(* Read only; Axis ID of the linked NC Axis *)
PROPERTY NcAxisId : UDINT
GET
NcAxisId := _AxisRef.NcToPlc.AxisId;
END_GET
END_PROPERTY

(* Read only; Axis ID of the linked NC Axis *)
PROPERTY NcAxisName : String(31)
GET
 NcAxisName := stAxisName;
END_GET
END_PROPERTY

METHOD ParamCheck : BOOL;
VAR_INST
  bTmp      : Bool;
  res       : Tc2_MC2.ST_McOutputs;
  nState    : DINT;
  stParaNr  : Tc2_MC2.MC_AxisParameter;
END_VAR

CASE nState 
OF
  0:
    ReadParameter(FALSE, stParaNr);
    bTmp              := FALSE;
    nState            := 1;
END_CASE
CASE nState 
OF
  1:
    IF NOT stDefaultAcceleration.bValid 
    THEN
      stParaNr        := AxisAcc;
      nState          := 10;

    ELSIF NOT stDefaultDeceleration.bValid 
    THEN
      stParaNr        := AxisDec;
      nState          := 10;

    ELSIF NOT stDefaultJerk.bValid 
    THEN
      stParaNr        := AxisJerk;
      nState          := 10;

    ELSIF NOT stHomingSearchVelo.bValid 
    THEN
      stParaNr        := AxisCalibrationVelocityForward;
      nState          := 10;

    ELSIF NOT stHomingVelo.bValid 
    THEN
      stParaNr        := AxisCalibrationVelocityBackward;
      nState          := 10;

    ELSIF NOT stMaxAcceleration.bValid 
    THEN
      stParaNr        := AxisMaximumAcceleration;
      nState          := 10;

    ELSIF NOT stMaxDeceleration.bValid 
    THEN
      stParaNr        := AxisMaximumDeceleration;
      nState          := 10;

    ELSIF NOT stMaxVelocity.bValid 
    THEN
      stParaNr        := AxisVeloMax;
      nState          := 10;

    ELSIF NOT stSwPosLimitNegative.bValid 
    THEN
      stParaNr        := AxisMinSoftPosLimit;
      nState          := 10;

    ELSIF NOT stSwPosLimitNegativeActive.bValid 
    THEN
      stParaNr        := AxisEnMinSoftPosLimit;
      nState          := 10;

    ELSIF NOT stSwPosLimitPositive.bValid 
    THEN
      stParaNr        := AxisMaxSoftPosLimit;
      nState          := 10;

    ELSIF NOT stSwPosLimitPositiveActive.bValid 
    THEN
      stParaNr        := AxisEnMaxSoftPosLimit;
      nState          := 10;

    ELSIF NOT stTargetPositionWindow.bValid 
    THEN
      stParaNr        := AxisTargetPositionWindow;
      nState          := 10;

    ELSE
      fbGetCurTaskIndex();
      _rCycleTime     := UDINT_TO_LREAL(_TaskInfo[fbGetCurTaskIndex.index].CycleTime)/10000.0;

      bTmp            := TRUE; // done
    END_IF
END_CASE
CASE nState 
OF
  10:
    bTmp              := FALSE;
    res               := ReadParameter(FALSE, stParaNr);
    nState            := 20;
END_CASE
CASE nState 
OF
  20:
    res               := ReadParameter(TRUE, stParaNr);
    IF res.Done
    THEN
      nState          := 30;
    END_IF

END_CASE
CASE nState 
OF
  30:
    nState                                := 0;
    CASE stParaNr 
    OF
      AxisEnMinSoftPosLimit: 
        stSwPosLimitNegativeActive.bValue := LREAL_TO_BOOL(fbReadParameter.Value);
        stSwPosLimitNegativeActive.bValid := TRUE;
    
      AxisEnMaxSoftPosLimit: 
        stSwPosLimitPositiveActive.bValue := LREAL_TO_BOOL(fbReadParameter.Value);
        stSwPosLimitPositiveActive.bValid := TRUE;
    
      AxisAcc: 
        stDefaultAcceleration.fValue      := fReadParamValue;
        stDefaultAcceleration.bValid      := TRUE;

      AxisDec: 
        stDefaultDeceleration.fValue      := fReadParamValue;
        stDefaultDeceleration.bValid      := TRUE;

      AxisJerk: 
        stDefaultJerk.fValue              := fReadParamValue;
        stDefaultJerk.bValid              := TRUE;

      AxisMaximumAcceleration : 
        stMaxAcceleration.fValue          := fReadParamValue;
        stMaxAcceleration.bValid          := TRUE;

      AxisMaximumDeceleration: 
        stMaxDeceleration.fValue          := fReadParamValue;
        stMaxDeceleration.bValid          := TRUE;

      AxisVeloMax: 
        stMaxVelocity.fValue              := fReadParamValue;
        fDefaultVelocity                  := stMaxVelocity.fValue * 0.1;
        stMaxVelocity.bValid              := TRUE;

      AxisMinSoftPosLimit: 
        stSwPosLimitNegative.fValue       := fReadParamValue;
        stSwPosLimitNegative.bValid       := TRUE;

      AxisMaxSoftPosLimit: 
        stSwPosLimitPositive.fValue       := fReadParamValue;
        stSwPosLimitPositive.bValid       := TRUE;

      AxisCalibrationVelocityForward: 
        stHomingSearchVelo.fValue         := fReadParamValue;
        stHomingSearchVelo.bValid         := TRUE;

      AxisCalibrationVelocityBackward: 
        stHomingVelo.fValue               := fReadParamValue;
        stHomingVelo.bValid               := TRUE;

      AxisTargetPositionWindow:
        stTargetPositionWindow.fValue     := fReadParamValue;
        stTargetPositionWindow.bValid     := TRUE;

    END_CASE

END_CASE

ParamCheck := bTmp;
END_METHOD

PROPERTY pAxisRef : POINTER TO AXIS_REF
GET
pAxisRef := ADR(_AxisRef);
END_GET
END_PROPERTY

PROPERTY Position : LREAL
GET
Position := _AxisRef.NcToPlc.ActPos;
END_GET
END_PROPERTY

{attribute '''NORMAL__COMMENT' := ' Will try to read a parameter from the NC axis; If the value is read, the Value is available at the ReadParamValue property.
  Refer to MC_ReadParameter Function Block in the Tc2_MC2 library; READMODE_ONCE is used as ReadMode '}
(* Will try to read a parameter from the NC axis; If the value is read, the Value is available at the ReadParamValue property.
  Refer to MC_ReadParameter Function Block in the Tc2_MC2 library; READMODE_ONCE is used as ReadMode *)
METHOD ReadParameter : Tc2_MC2.ST_McOutputs
VAR_INPUT
  Execute           : BOOL;
  (* Number of the parameter to be read. Refer to the MC_AxisParameter type defined at Tc2_MC2 library *)
  {attribute '''NORMAL__COMMENT' := ' Number of the parameter to be read. Refer to the MC_AxisParameter type defined at Tc2_MC2 library '}
  ParameterNumber   : Tc2_MC2.MC_AxisParameter;
END_VAR
VAR_INST
  res               : Tc2_MC2.ST_McOutputs;
  nState            : DINT;
END_VAR

CASE nState OF
  0:
    IF Execute
    THEN
      memset(ADR(res),0,SIZEOF(res));
      res.Busy                          := TRUE;

      fbReadParameter.ParameterNumber   := ParameterNumber;
      fbReadParameter.Enable            := FALSE;

      nState                            := 10;
    END_IF
END_CASE
CASE nState OF
  10:
    fbReadParameter.Enable              := TRUE;

    IF fbReadParameter.Valid
    THEN
      fbReadParameter.Enable            := FALSE;
      nState                            := 20;
    ELSE
      IF fbReadParameter.Error
      THEN
        res.ErrorID                     := fbWriteParameter.ErrorID;

        stMsg.eType                     := E_MessageType.eMessageError;
        stMsg.eDevice                   := e_Device.Axis + TO_DINT(_AxisRef.NcToPlc.AxisId);
        stMsg.eSubdevice                := e_SubDevice.fbReadParameter;
        stMsg.iErrorNumber              := fbReadParameter.ErrorID;

        f_MessageSet(stMsg);
        MsgAdd(stMsg);

        fbReadParameter.Enable          := FALSE;
        nState                          := 99;
      END_IF
    END_IF
END_CASE
CASE nState OF
  20:
    res.Busy                            := FALSE;
    res.Done                            := TRUE;

  99:
    res.Busy                            := FALSE;
    res.Error                           := TRUE;
END_CASE

fbReadParameter(Axis                    := _AxisRef, 
                ParameterNumber         := ParameterNumber, 
                ReadMode                := Tc2_MC2.READMODE_ONCE, 
                Value                   => fReadParamValue);

IF NOT Execute
THEN
  memset(ADR(res),0,SIZEOF(res));
  nState                                := 0;
END_IF

ReadParameter := res;
END_METHOD

(* Read only; Returns the value from the last successful read by ReadParameter methode *)
PROPERTY ReadParamValue : LREAL
GET
ReadParamValue := fReadParamValue;
END_GET
END_PROPERTY

(* Speed override factor in percent [%] to all movements. Refer to MC_Power Function Block in the Tc2_MC2 library *)
PROPERTY SpeedOverride : LREAL
GET
SpeedOverride := fbPower.Override;
END_GET
SET
fbPower.Override := SpeedOverride;
END_SET
END_PROPERTY

PROPERTY StartUpDone : BOOL
GET
StartUpDone := _bStartUp;
END_GET
END_PROPERTY

PROPERTY StartUpError : Bool
GET
StartUpError := _bStartUpError;
END_GET
END_PROPERTY

(* Read only; Initiates read the actual Axis status; returns the Status of the last performed read *) 
PROPERTY Status : Tc2_MC2.ST_AxisStatus
GET
Status := _AxisRef.Status;
END_GET
END_PROPERTY

METHOD Stop : Tc2_MC2.ST_McOutputs
VAR_INPUT
  Execute   : BOOL;
END_VAR
VAR_INST
  res       : Tc2_MC2.ST_McOutputs;
  nState    : DINT;
  fUsedDec,
  fUsedJerk : LREAL;
  itmp      : DINT;
END_VAR
CASE nState OF
  0:
    IF Execute
    THEN
      memset(ADR(res),0,SIZEOF(res));
      memset(ADR(itmp),0,SIZEOF(itmp));
      res.Busy                := TRUE;

      fUsedDec                := stDefaultDeceleration.fValue;
      fUsedJerk               := stDefaultJerk.fValue;

      fbStop(Axis             := _AxisRef,  
             Execute          := FALSE, 
             Deceleration     := fUsedDec, 
             Jerk             := fUsedJerk);

      fbReset(Axis            := _AxisRef, 
              Execute         := FALSE);

      nState := 10;
    END_IF
END_CASE
CASE nState OF
  10:
    fbStop(Axis               := _AxisRef, 
           Execute            := TRUE);

    IF fbStop.Done
    THEN
      fbStop(Axis             := _AxisRef, 
             Execute          := FALSE);

      nState := 20;

    ELSE
      IF fbStop.Error
      THEN
        res.ErrorID           := fbStop.ErrorID;

        stMsg.eType           := E_MessageType.eMessageError;
        stMsg.eDevice         := e_Device.Axis + UDINT_TO_DINT(_AxisRef.NcToPlc.AxisId);
        stMsg.eSubdevice      := e_SubDevice.fbStop;
        stMsg.iErrorNumber    := fbStop.ErrorID;
        f_MessageSet(stMsg);
        MsgAdd(stMsg);

        fbReset(Axis          := _AxisRef, 
                Execute       := TRUE);

        nState := 98;

      ELSIF NOT _AxisRef.Status.Stopping
      THEN
        itmp := itmp +1;
        // todo: faststop?
      END_IF
    END_IF
END_CASE
CASE nState OF
  20:
    res.Busy := FALSE;
    res.Done := TRUE;

  98:
    fbStop(Axis               := _AxisRef, 
           Execute            := FALSE);

    fbReset(Axis              := _AxisRef, 
            Execute           := FALSE);
    nState := 99;

END_CASE
CASE nState OF
  99:
    res.Busy                  := FALSE;
    res.Error                 := TRUE;
END_CASE

IF NOT Execute
THEN
  memset(ADR(res),0,SIZEOF(res));
  nState                      := 0;
END_IF

Stop := res;
END_METHOD

PROPERTY Version : STRING
(* ToDo:
- Testen
*)
GET
Version := '1.0';
(*
  0.1   09.2016 MR  Erste Version des Achsbausteins als OOP Wrapper der MC Bausteine; Die Funktionen können meißt (Außnahme: Jog) durch einen einmaliger Methodenaufruf angestossen werden;
            der weitere Aufruf erfolgt dann automatisch über den zyklischen Aufruf der FB Instanz und die interne Methode CyclicCallOnBusy. Die FB Instanz muss immer zyklisch 
            aufgerufen werden.
            
  1.0
  2022 06 30
  HAUD
  - 
  - cyclic method calls required
  - motion methods contain VAR_INST (fixed procedure, no race conditions)
  - Motion Parameter as properties (input from stCtrl by AxisController)
  - cyclic ca

*)
END_GET
END_PROPERTY

{attribute '''NORMAL__COMMENT' := ' Will try to write a parameter from the NC axis; Refer to MC_WriteParameter Function Block in the Tc2_MC2 library '}
(* Will try to write a parameter from the NC axis; Refer to MC_WriteParameter Function Block in the Tc2_MC2 library *)
METHOD WriteParameter : Tc2_MC2.ST_McOutputs
VAR_INPUT
  Execute   : BOOL;
  (* Number of the parameter to be written. Refer to the MC_AxisParameter type defined at Tc2_MC2 library *)
  {attribute '''NORMAL__COMMENT' := ' Number of the parameter to be written. Refer to the MC_AxisParameter type defined at Tc2_MC2 library '}
  ParameterNumber : Tc2_MC2.MC_AxisParameter;
  (* defines the value to be written to the parameter *)
  {attribute '''NORMAL__COMMENT' := ' defines the value to be written to the parameter '}
  Value : LREAL;
END_VAR
VAR_INST
  res       : Tc2_MC2.ST_McOutputs;
  nState    : DINT;
END_VAR

CASE nState OF
  0:
    IF Execute
    THEN
      memset(ADR(res),0,SIZEOF(res));

      res.Busy                                := TRUE;

      fbWriteParameter.ParameterNumber        := ParameterNumber;

      fbWriteParameter(Axis                   := _AxisRef, 
                       Execute                := FALSE);
 
      nState                                  := 10;
    END_IF
END_CASE
CASE nState OF
  10:
    fbWriteParameter.Execute                  := TRUE;

    IF fbWriteParameter.Done
    THEN
      nState                                  := 20;

      CASE fbWriteParameter.ParameterNumber 
      OF
        AxisEnMinSoftPosLimit: 
          stSwPosLimitNegativeActive.bValue   := TO_BOOL(Value);

        AxisEnMaxSoftPosLimit: 
          stSwPosLimitPositiveActive.bValue   := TO_BOOL(Value);

        AxisAcc: 
          stDefaultAcceleration.fValue        := Value;

        AxisDec: 
          stDefaultDeceleration.fValue        := Value;

        AxisJerk: 
          stDefaultJerk.fValue                := Value;

        AxisMaximumAcceleration : 
          stMaxAcceleration.fValue            := Value;

        AxisMaximumDeceleration: 
          stMaxDeceleration.fValue            := Value;

        AxisVeloMax: 
          stMaxVelocity.fValue                := Value;

        AxisMinSoftPosLimit: 
          stSwPosLimitNegative.fValue         := Value;

        AxisMaxSoftPosLimit: 
          stSwPosLimitPositive.fValue         := Value;

        AxisCalibrationVelocityForward: 
          stHomingSearchVelo.fValue           := Value;

        AxisCalibrationVelocityBackward: 
          stHomingVelo.fValue                 := Value;

        AxisTargetPositionWindow:
          stTargetPositionWindow.fValue       := Value;
      END_CASE
    ELSE
      IF fbWriteParameter.Error
      THEN
        res.Busy                              := FALSE;
        res.Error                             := TRUE;
        res.ErrorID                           := fbWriteParameter.ErrorID;

        stMsg.eType                           := E_MessageType.eMessageError;
        stMsg.eDevice                         := e_Device.Axis + TO_DINT(_AxisRef.NcToPlc.AxisId);
        stMsg.eSubdevice                      := e_SubDevice.fbWriteParameter;
        stMsg.iErrorNumber                    := fbWriteParameter.ErrorID;

        fbWriteParameter.Execute              := FALSE;

        f_MessageSet(stMsg);
        MsgAdd(stMsg);

        nState                                := 99;
      END_IF
    END_IF
END_CASE
CASE nState OF
  20:
    res.Busy                                  := FALSE;
    res.Done                                  := TRUE;

  99:
    res.Busy                                  := FALSE;
    res.Error                                 := TRUE;

END_CASE


IF NOT Execute
THEN
  memset(ADR(res),0,SIZEOF(res));

  fbWriteParameter.Execute                    := FALSE;
  nState                                      := 0;
END_IF


fbWriteParameter(Axis                         := _AxisRef, 
                 ParameterNumber              := ParameterNumber, 
                 Value                        := Value, 
                 Done                         => WriteParameter.Done, 
                 Busy                         => WriteParameter.Busy, 
                 Error                        => WriteParameter.Error, 
                 ErrorID                      => WriteParameter.ErrorID);


WriteParameter := res;
END_METHOD

END_FUNCTION_BLOCK

// ---- POUs/MSG/f_MessageSet.TcPOU
FUNCTION f_MessageSet : BOOL
VAR_INPUT
  stMessage   : ST_Message;
END_VAR
VAR
  uiIndex   : INT;
  uiFound   : INT;
END_VAR

stMessage.tTime := GVL_AXIS_CTRL.gsLocalTime;

FOR uiIndex := 1 TO GVL_AXIS_CTRL.gciMaxMessage
DO
  IF (GVL_AXIS_CTRL.gatMessages[uiIndex].eType = e_MessageType.eMessageEmpty)
  THEN
    GVL_AXIS_CTRL.gatMessages[uiIndex] := stMessage;
    GVL_AXIS_CTRL.giMsgIndex := uiIndex;
    EXIT;
  END_IF
END_FOR

IF (stMessage.eType = E_MessageType.eMessageError)
THEN
  GVL_AXIS_CTRL.giErrorIndex := GVL_AXIS_CTRL.giErrorIndex + 1;
END_IF

END_FUNCTION

// ---- POUs/_FunctionBlocks/fb_ResetSercos.TcPOU
FUNCTION_BLOCK fb_ResetSercos
VAR_INPUT
	bExecute  : BOOL;
	eDevice		: e_Device;
	p_AxisRef	: POINTER TO Tc2_MC2.AXIS_REF;
END_VAR
VAR_OUTPUT
	stMcOutput : ST_McOutputs;
END_VAR
VAR
	diStep			: DINT;
	tonDelay		: ton;
	_stMessage	: ST_Message;
	fbResetSercos		: FB_SoEReset;
	iRepeat			: INT;
END_VAR

IF NOT bExecute
THEN
	stMcOutput.Active := FALSE;
	stMcOutput.Done := FALSE;
	diStep := 0;
END_IF

IF bExecute AND diStep = 0
THEN
	diStep := 10;
END_IF

IF p_AxisRef = 0
THEN
	RETURN;
END_IF

CASE diStep OF

	0:
		iRepeat := 0;
		tonDelay(IN:= FALSE);
		fbResetSercos(
			NetId:= , 
			Execute:= FALSE, 
			Timeout:= , 
			Axis:= p_AxisRef^, 
			Busy=> , 
			Error=> , 
			AdsErrId=> , 
			SercosErrId=> );

	10:
		stMcOutput.Active := TRUE;
		tonDelay(PT:= T#1500MS, IN:= TRUE);
		fbResetSercos(
			NetId:= , 
			Execute:= TRUE, 
			Timeout:= , 
			Axis:= p_AxisRef^, 
			Busy=> , 
			Error=> , 
			AdsErrId=> , 
			SercosErrId=> );

		IF NOT fbResetSercos.Busy
		THEN
			diStep := 20;
		END_IF

		IF tonDelay.Q AND p_AxisRef^.NcToPlc.StateDWord.28
		THEN
			iRepeat := iRepeat + 1;
			tonDelay(IN:= FALSE);
			fbResetSercos(
				NetId:= , 
				Execute:= FALSE, 
				Timeout:= , 
				Axis:= p_AxisRef^, 
				Busy=> , 
				Error=> , 
				AdsErrId=> , 
				SercosErrId=> );
		END_IF
 

	20:
		stMcOutput.Done := TRUE;

		IF NOT bExecute
		THEN
			fbResetSercos(Execute:= FALSE, Axis:= p_AxisRef^);
			memset(ADR(stMcOutput), 0, SIZEOF(stMcOutput));
			diStep :=0;
		END_IF
END_CASE

stMcOutput.Busy 		:= fbResetSercos.Busy;
stMcOutput.Error 		:= fbResetSercos.Error;
stMcOutput.ErrorID 	:= fbResetSercos.SercosErrId;

// push error
IF fbResetSercos.Execute AND fbResetSercos.Error THEN
	_stMessage.eDevice := eDevice;
	_stMessage.eSubdevice := e_SubDevice.fbResetSercos;
	_stMessage.iErrorNumber := fbResetSercos.SercosErrId;
	_stMessage.tTime := GVL_AXIS_CTRL.gsLocalTime;

	f_MessageSet(_stMessage);
END_IF

END_FUNCTION_BLOCK

// ---- POUs/_FunctionBlocks/FB_XenaxEtherCATHoming.TcPOU
FUNCTION_BLOCK FB_XenaxEtherCATHoming
VAR_INPUT

  bExecute        :BOOL;

  bAbort          :BOOL:=FALSE;
END_VAR
VAR_IN_OUT
  Axis            :AXIS_REF;
END_VAR
VAR_OUTPUT
  Done            :BOOL;    (* successfully done *)
  Busy            :BOOL;    (* busy, not in initial state *)
  Error           :BOOL;    (* Error flag *)
  ErrorId         :UDINT;   (* Error code *)
END_VAR

VAR CONSTANT

END_VAR
VAR
  fbCoEReadParameter        : FB_EcCoESdoRead;
  fbCoEWriteParameter       : FB_EcCoESdoWrite;
  WriteNC                   : ADSWRITE;
  ReadNC                    : ADSREAD;
  ResetAxis                 : MC_Reset;

  abySend,
  abyReceive                : ARRAY[0..10] OF BYTE;




  state                     : INT;
  ErrorState                : INT;   (* state where the latest error occured *)
  LagDistanceMonitoring     : UINT;
  SavedLagDistanceMonitoring: UINT;
  Trigger                   : R_TRIG;
  Delay                     : TON;
  ExecuteOffTrigger         : F_TRIG;
  NcReferenceFlag           : DWORD;

  fbGetAmsNetID             : FB_GetAxisAmsAddr;

  sEtherCATNetId            : STRING; (*Master Ethercat AMS Adress *)
  nSlaveAddr                : INT := 1001;  (* Slave adress in system manager *)

  lrPosBefore               : LREAL;
  lrPosAfter                : LREAL;
END_VAR

(*****************************************************************************************************)
(*  Jenny Science AG                              *)
(*                                    *)
(*  Date    : 22.08.2011                      *)
(*****************************************************************************************************)
(*  Version   : 1.51                            *)
(*****************************************************************************************************)
(*  Description : Exemple for Homing Programm for Xenax Xvi75v8     *)
(*                                            1.51 *smal correction on step 62                                     *)
(*                                            1.5 Control that Homing start correctly                                    *)
(*                                            1.4 Wait Homing Done with Object 2006 Bit 1                                   *)
(*                                            1.3 Resolution of negativ position after Homing                              *)
(*****************************************************************************************************)
ExecuteOffTrigger(CLK:=bExecute);



CASE state OF
(*************************************************************************************************************************)
 (* initial state, wait for trigger *)
  0 :
    Busy := FALSE;
    Trigger( CLK:=bExecute );
    IF Trigger.Q THEN
      state := 10;
    END_IF

  10:
    fbGetAmsNetID(  sNetId:= '',
            iAxisId:= TO_UINT(Axis.NcToPlc.AxisId),
            bExecute := TRUE);
    IF NOT fbGetAmsNetID.bBusy AND NOT fbGetAmsNetID.bError THEN
      sEtherCATNetId  := fbGetAmsNetID.AxisNetId;
      nSlaveAddr    := TO_INT(fbGetAmsNetID.AxisPort);

      fbGetAmsNetID(  sNetId:= '',
              iAxisId:= TO_UINT(Axis.NcToPlc.AxisId),
              bExecute := FALSE);
      Busy := TRUE;
      Done := FALSE;
      Error := FALSE;
      ErrorID := 0;
      ErrorState := 0;
      WriteNC( WRITE:=FALSE );
      ReadNC( READ:=FALSE );
      ResetAxis(Execute:=FALSE, Axis:=Axis);
      Delay(IN:=FALSE);
      state := 15;
  END_IF
(* Read lag distance monitoring *)
  15 :
    ReadNC  (NETID:='' , PORT:=AMSPORT_R0_NC , IDXGRP:=NCIDXG_AXPARMS+DWORD_TO_UINT(Axis.NcToPlc.AxisId) , IDXOFFS:=16#20010 , LEN:=SIZEOF(SavedLagDistanceMonitoring) , DESTADDR:=ADR(SavedLagDistanceMonitoring) , READ:=TRUE , TMOUT:=T#1S);
    IF NOT ReadNC.Busy AND NOT ReadNC.Err THEN
      ReadNC( READ:=FALSE );
      state := 20;
    END_IF
(* Desable lag distance monitoring  *)
  20 :
    LagDistanceMonitoring := 0;
    WriteNC(NETID:='' , PORT:=AMSPORT_R0_NC , IDXGRP:=NCIDXG_AXPARMS+DWORD_TO_UINT(Axis.NcToPlc.AxisId) , IDXOFFS:=16#20010 , LEN:=SIZEOF(LagDistanceMonitoring) , SRCADDR:=ADR(LagDistanceMonitoring) , WRITE:=TRUE , TMOUT:=T#1s);
    IF NOT WriteNC.Busy AND NOT WriteNC.Err THEN
      WriteNC( WRITE:=FALSE );
      state := 25;
    END_IF
(*************************************************************************************************************************)
 (* disable NC reference flag *)
  25 :
    NcReferenceFlag := 0;
    WriteNC(NETID:='' , PORT:=AMSPORT_R0_NC , IDXGRP:=NCIDXG_AXFUNCS+DWORD_TO_UINT(Axis.NcToPlc.AxisId) , IDXOFFS:=16#1B , LEN:=SIZEOF(NcReferenceFlag) , SRCADDR:=ADR(NcReferenceFlag) , WRITE:=TRUE , TMOUT:=T#1s);
    IF NOT WriteNC.Busy AND NOT WriteNC.Err THEN
      WriteNC( WRITE:=FALSE );
      state := 30;
    END_IF
(*************************************************************************************************************************)
(* Set OpMode 6 -> Start Homing *)
  30 :
    fbCoEWriteParameter.nIndex    := 16#6060;
    fbCoEWriteParameter.nSubIndex := 0;
    abySend[0]            :=6;
    fbCoEWriteParameter.cbBufLen    :=1;
    fbCoEWriteParameter.bExecute  := TRUE;
    state := 40;
(*************************************************************************************************************************)
  40 :
    IF NOT fbCoEWriteParameter.bBusy THEN
      fbCoEWriteParameter.bExecute  := FALSE;
        state := 50;
    END_IF;

(*************************************************************************************************************************)
(* Control that the Homing method is setting into the Xenax , after 500ms                                                               *)
  50 :

    Delay(IN:=TRUE , PT:=t#500ms );
    IF Delay.Q THEN
      fbCoEReadParameter.nIndex   := 16#6061;
      fbCoEReadParameter.nSubIndex  := 0;
      fbCoEReadParameter.cbBufLen   := 1;
      fbCoEReadParameter.bExecute   := TRUE;
      Delay(IN:=FALSE);
      state := 51;
    END_IF

(*************************************************************************************************************************)
 (*  if the method is correctly setted goes next (step 70), else repeat the setting method *)
  51:

    IF NOT fbCoEReadParameter.bBusy THEN

      fbCoEReadParameter.bExecute   := FALSE;

      IF abyReceive[0] = 6 THEN
        state := 70;
      ELSE
        state := 60;
      END_IF
    END_IF;

(*************************************************************************************************************************)
 (* Repeat the Homing started Method *)
(* Set OpMode 6 -> 0*)
  60 :
    fbCoEWriteParameter.nIndex    := 16#6060;
    fbCoEWriteParameter.nSubIndex := 0;
    abySend[0]            :=0;
    fbCoEWriteParameter.cbBufLen    :=1;
    fbCoEWriteParameter.bExecute  := TRUE;
    state := 61;
  61 :
    IF NOT fbCoEWriteParameter.bBusy THEN
      fbCoEWriteParameter.bExecute  := FALSE;
        state := 62;
    END_IF;
(*************************************************************************************************************************)
(* Wait Time *)
  62 :
    Delay(IN:=TRUE , PT:=t#500ms );
    IF Delay.Q THEN
      Delay(IN:=FALSE);
      state := 30;
    END_IF

(*************************************************************************************************************************)
(*Read Axis referenced after 200ms *)
  70 :

    Delay(IN:=TRUE , PT:=t#200ms );
    IF Delay.Q THEN
      fbCoEReadParameter.nIndex   := 16#2006;
      fbCoEReadParameter.nSubIndex  := 0;
      fbCoEReadParameter.cbBufLen   :=4;
      fbCoEReadParameter.bExecute   := TRUE;
      Delay(IN:=FALSE);
      state := 80;
    END_IF

(*************************************************************************************************************************)
 (* Wait Achse referenced *)
  80:

    IF NOT fbCoEReadParameter.bBusy THEN

      fbCoEReadParameter.bExecute   := FALSE;

      IF abyReceive[0].1 THEN
        lrPosBefore := Axis.NcToPlc.ActPos;
        state := 90;
      ELSE
        state := 70;

      END_IF
END_IF;

(*************************************************************************************************************************)
 (* Wait some time before resetting the TwinCAT axis position *)
  90 :
    Delay(IN:=TRUE , PT:=t#200ms );
    IF Delay.Q THEN
      lrPosAfter := Axis.NcToPlc.ActPos;

      Delay(IN:=FALSE);
      state := 110;
    END_IF

(*************************************************************************************************************************)
 (* Reset *)
  110:
    ResetAxis(Execute:=TRUE , Axis:=Axis );
    IF ResetAxis.Done OR ResetAxis.Error THEN
      ResetAxis(Execute:=FALSE, Axis:=Axis);
      state :=200;
    END_IF
(*************************************************************************************************************************)
(* set lag distance monitoring to its original value *)
  200 :
    WriteNC(NETID:='' , PORT:=AMSPORT_R0_NC , IDXGRP:=NCIDXG_AXPARMS+DWORD_TO_UINT(Axis.NcToPlc.AxisId) , IDXOFFS:=16#20010 , LEN:=SIZEOF(SavedLagDistanceMonitoring) , SRCADDR:=ADR(SavedLagDistanceMonitoring) , WRITE:=TRUE , TMOUT:=T#1s);
    IF NOT WriteNC.Busy AND NOT WriteNC.Err THEN
      WriteNC( WRITE:=FALSE );
      state := 210;
    END_IF
(*************************************************************************************************************************)
 (* Enable NC reference flag *)
  210 :
    NcReferenceFlag := 1;
    WriteNC(NETID:='' , PORT:=AMSPORT_R0_NC , IDXGRP:=NCIDXG_AXFUNCS+DWORD_TO_UINT(Axis.NcToPlc.AxisId) , IDXOFFS:=16#1B , LEN:=SIZEOF(NcReferenceFlag) , SRCADDR:=ADR(NcReferenceFlag) , WRITE:=TRUE , TMOUT:=T#1s);
    IF NOT WriteNC.Busy AND NOT WriteNC.Err THEN
      WriteNC( WRITE:=FALSE );
      state := 220;
    END_IF
(*************************************************************************************************************************)
(* Set OpMode 8 *)
  220 :
    fbCoEWriteParameter.nIndex    := 16#6060;
    fbCoEWriteParameter.nSubIndex := 0;
    abySend[0]            :=8;
    fbCoEWriteParameter.cbBufLen    :=1;
    fbCoEWriteParameter.bExecute  := TRUE;
    state := 230;
(*************************************************************************************************************************)
(* Wait end*)
  230 :
  IF NOT fbCoEWriteParameter.bBusy THEN
    fbCoEWriteParameter.bExecute  := FALSE;
      state := 240;
  END_IF;
(*************************************************************************************************************************)
(* Wait 200ms*)
  240 :
    Delay(IN:=TRUE , PT:=t#200ms );
    IF Delay.Q THEN
      Delay(IN:=FALSE);
      state := 1000;
    END_IF


(***************************************************************************************************************)
(*ABORT*)
(*************************************************************************************************************************)
(*************************************************************************************************************************)
 (* Reset *)
  400:
    ResetAxis(Execute:=TRUE , Axis:=Axis);
    IF ResetAxis.Done OR ResetAxis.Error THEN
      ResetAxis(Execute:=FALSE, Axis:=Axis);
      state :=410;
    END_IF
(*************************************************************************************************************************)
(* set lag distance monitoring to its original value *)
  410 :
    LagDistanceMonitoring := 0;
    WriteNC(NETID:='' , PORT:=AMSPORT_R0_NC , IDXGRP:=NCIDXG_AXPARMS+DWORD_TO_UINT(Axis.NcToPlc.AxisId) , IDXOFFS:=16#20010 , LEN:=SIZEOF(SavedLagDistanceMonitoring) , SRCADDR:=ADR(SavedLagDistanceMonitoring) , WRITE:=TRUE , TMOUT:=T#1s);
    IF NOT WriteNC.Busy AND NOT WriteNC.Err THEN
      WriteNC( WRITE:=FALSE );
      state := 420;
    END_IF
(*************************************************************************************************************************)
(* Set OpMode 8 *)
  420 :
    fbCoEWriteParameter.nIndex    := 16#6060;
    fbCoEWriteParameter.nSubIndex := 0;
    abySend[0]            :=8;
    fbCoEWriteParameter.cbBufLen    :=1;
    fbCoEWriteParameter.bExecute  := TRUE;
    state := 430;
(*************************************************************************************************************************)
(* Wait end of Set OpMode 8 *)
  430 :
  IF NOT fbCoEWriteParameter.bBusy THEN
    fbCoEWriteParameter.bExecute  := FALSE;
      state := 1000;
  END_IF;
(*************************************************************************************************************************)
(* End *)
  1000 :
    Done:=TRUE;
    Busy:=FALSE;
    IF NOT bExecute AND NOT bAbort THEN
      state:=0;
      Done:=FALSE;
    END_IF;
END_CASE

(* check for errors *)
IF state <> 0 THEN
  IF WriteNC.ERR AND WriteNC.WRITE THEN
    Error := TRUE;
    ErrorId := WriteNC.ErrId;
  ELSIF ReadNC.ERR AND ReadNC.READ THEN
    Error := TRUE;
    ErrorId := ReadNc.ErrId;
  END_IF
  IF Error THEN
    ErrorState := state;
    state := 0;
  END_IF
END_IF


fbCoEReadParameter(   sNetId    := sEtherCATNetId,
            nSlaveAddr  := TO_UINT(nSlaveAddr),
            tTimeout    := T#500ms,
            pDstBuf   :=ADR(abyReceive));

fbCoEWriteParameter(    sNetId    := sEtherCATNetId,
            nSlaveAddr  := TO_UINT(nSlaveAddr),
            pSrcBuf   :=ADR(abySend),
            tTimeout    := T#500ms);

END_FUNCTION_BLOCK

// ---- POUs/_FunctionBlocks/cam/FB_CamIn_empty.TcPOU
FUNCTION_BLOCK FB_CamIn_empty
VAR_INPUT
  Master            : REFERENCE TO Tc2_MC2.AXIS_REF;
  Slave             : REFERENCE TO Tc2_MC2.AXIS_REF; 
  Execute           : BOOL;
  MasterOffset      : REAL; 
  SlaveOffset       : REAL; 
  MasterScaling     : REAL;
  SlaveScaling      : REAL;
  StartMode         : INT;
  CamTableID        : UDINT;
END_VAR
VAR_OUTPUT
  Busy              : BOOL;
  Error             : BOOL;
  Done              : BOOL;
  InSync            : BOOL;
  ErrorId           : UDINT;
END_VAR
VAR
END_VAR


Error   := TRUE;
ErrorId := 9999; // function is not activated by compiler def CAM

END_FUNCTION_BLOCK

// ---- POUs/_FunctionBlocks/cam/FB_CamOut_Empty.TcPOU
FUNCTION_BLOCK FB_CamOut_Empty
VAR_INPUT
  Slave             : REFERENCE TO Tc2_MC2.AXIS_REF;
  Execute           : BOOL;
END_VAR
VAR_OUTPUT
  Busy              : BOOL;
  Error             : BOOL;
  Done              : BOOL;
  ErrorId           : UDINT;
END_VAR
VAR
END_VAR


Error   := TRUE;
ErrorId := 9999; // function is not activated by compiler def CAM

END_FUNCTION_BLOCK

// ---- POUs/MAPPING/MAPPING_out.TcPOU
PROGRAM MAPPING_out
VAR CONSTANT
{IF defined (AXIS_MAP)}
  {info 'MAPPING_out - ACTIVE'}
  bBypassMapping    : BOOL  := FALSE;
{ELSE}
  bBypassMapping    : BOOL  := TRUE;
{END_IF}
END_VAR
VAR
  AxisState         : U_AXIS_STATE;
  AxisInfo          : U_AXIS_INFO;
  AxisParameterRd   : U_AXIS_NC_PARAMETER;

  nAxis             : INT;
END_VAR

IF bBypassMapping THEN RETURN; END_IF

FOR nAxis := 1 TO GVL_AXIS_CTRL.gciMaxAxis
DO
  AxisState.stState[nAxis]        := GVL_AXIS_CTRL.gstAxisControl[nAxis].FromPlc;
  AxisInfo.stState[nAxis]         := GVL_AXIS_CTRL.gfbAxisController[nAxis].StatusCompact;

  AxisParameterRd.stState[nAxis]  := GVL_AXIS_CTRL.gstAxisParam[nAxis];
END_FOR

END_PROGRAM

// ---- POUs/NCI/FB_Ctrl_NciChannel.TcPOU
(*
-------------------------------------------------------------------------------
	NCI Channel Control

  2020/05/20  HAUD  0.1     kinematic and NCI separation
  2022/10/22  HAUD  0.2     PLC_OPEN_DRIVE adoption
-------------------------------------------------------------------------------
*)

// This SOFTWARE is provided as an Exemple by THE PROVIDER "as is" and "with all faults." THE PROVIDER makes no 
// representations or warranties of any kind concerning the safety, suitability, lack of viruses, inaccuracies, 
// typographical errors, or other harmful components of this SOFTWARE. There are inherent dangers in the use of 
// any software, and you are solely responsible for determining whether this SOFTWARE is compatible with your 
// equipment and other software installed on your equipment. You are also solely responsible for the protection 
// of your equipment and backup of your data, and THE PROVIDER will not be liable for any damages you may suffer 
// in connection with using, modifying, or distributing this SOFTWARE.

FUNCTION_BLOCK FB_Ctrl_NciChannel IMPLEMENTS I_Nci_Ctrl
VAR
  _eCmd                 : e_Ctrl_NciCommand;

  _sState                : STRING;
  _nErrorId              : UDINT;
  _bError                : BOOL;

  _fPathVelo             : LREAL;
  _nBlockNo              : UDINT;
  _sProgLine             : STRING(100); 
  _nMFunc                : INT;
  _eState                : e_Ctrl_NciCommand;
  _uiStateItp            : UINT;



  _stMsg                 : ST_Message;
  _ChannelDevice         : e_Device := e_Device.NciChannelCtrl;

  _eCmdState,
  _eCmdExec,
  _eCmdExecOld,
  _eCmdOld,
  _eCmdActive            : e_Ctrl_NciCommand;

  _sCmd,
  _sCmdOld,
  _sCmdExec              : STRING(256);

  _nState,
  _nStateSS1             : DINT;

{IF defined (WIN)}
  _sProg                : STRING(255) := 'C:\TwinCAT\Mc\Nci\Test_GST.nc';
{ELSE}
  _sProg                : STRING(255) := '/usr/local/etc/TwinCAT/Mc/Nci/Test_GST.nc';
{END_IF}

  _stMFuncCyclic        : ST_Ctrl_NciMFuncCycle;

  _nChnId               : UINT;
  // R[] Params used in G-Code
  // R[0..899]    local namespace of Channel
  // R[900..999]  global namespace of NC
  _iri,
  _irc,
  _iRParamIndex,
  _iRParamCount         : DINT;

  _rRParamsRead,
  _rRParamsWrite        : ARRAY [0..GVL_NCI.cRParamCount] OF LREAL;

//MCS-Axes
  _ipMcsAxis            : ARRAY[1..GVL_NCI.cMcAxisCount] OF I_McAxis;
  _iMcCount,
  _iMcCountConfigured   : DINT;
  _bMcAxisMismatch      : BOOL;

//Aux-Axes
  _ipAuxAxis            : ARRAY[1..GVL_NCI.cAuxAxisCount] OF I_McAxis;
  _iAuxCount,
  _iAuxCountConfigured  : DINT;
  _bAuxAxisMismatch     : BOOL;


  _bErrorCyclicChecks   : BOOL;

  _mdx,
  _adx                  : UINT;
  _hr                   : HRESULT;

  _fbNciChannel         : FB_NciChannel;
  _ipNciChannel         : I_NciChannel;

END_VAR

ACTION Channel_BuildGroup:
CASE _nState OF
  0:
    _hr                       := S_FALSE;
    _nState                   := 10;
END_CASE
CASE _nState OF
  10:
    _eCmdActive               := eCmd + e_Ctrl_NciCommand.CMD_BUSY;
    _eCmdExec                 := e_Ctrl_NciCommand.CMD_BUSY;

    _ipNciChannel.I_AuxAxis   := _ipAuxAxis;
    _ipNciChannel.I_McAxis    := _ipMcsAxis;

    _hr                       := _ipNciChannel.BuildGroup(FALSE);

    _nState                   := 20;
END_CASE
CASE _nState OF
  20:
    _hr                       := _ipNciChannel.BuildGroup(TRUE);

    IF (_hr = S_OK)
    THEN
      _hr                     := _ipNciChannel.BuildGroup(FALSE);
      _nState                 := 100;
    ELSE
      IF (_hr > S_FALSE)
      THEN
        _hr                   := _ipNciChannel.BuildGroup(FALSE);
        _nState               := 900;
      END_IF
    END_IF
END_CASE
CASE _nState OF
  100:
    _eCmdActive               := eCmd + e_Ctrl_NciCommand.CMD_DONE;
    _eCmdExec                 := e_Ctrl_NciCommand.CMD_DONE;
END_CASE
CASE _nState OF
  900:
    _eCmdActive               := eCmd + e_Ctrl_NciCommand.CMD_ERROR;
    _eCmdExec                 := e_Ctrl_NciCommand.CMD_ERROR;
END_CASE
END_ACTION

ACTION Channel_ClearGroup:
CASE _nState OF
  0:
    _ipNciChannel.pNciChannelRef^.PlcToNc.MFuncGranted := 1;
    _hr                       := S_FALSE;
    _nState                   := 10;

  10:
    _ipNciChannel.pNciChannelRef^.PlcToNc.MFuncGranted := 0;
    _eCmdActive               := eCmd + e_Ctrl_NciCommand.CMD_BUSY;
    _eCmdExec                 := e_Ctrl_NciCommand.CMD_BUSY;

    _ipNciChannel.I_AuxAxis   := _ipAuxAxis;
    _ipNciChannel.I_McAxis    := _ipMcsAxis;

    _hr                       := _ipNciChannel.ClearGroup(FALSE);

    _nState                   := 20;


  20:
    _ipNciChannel.pNciChannelRef^.PlcToNc.MFuncGranted := 1;
    _hr                       := _ipNciChannel.ClearGroup(TRUE);

    IF (_hr = S_OK)
    THEN
      _hr                     := _ipNciChannel.ClearGroup(FALSE);
      _nState                 := 100;
    ELSE
      IF (_hr > S_FALSE)
      THEN
        _hr                   := _ipNciChannel.ClearGroup(FALSE);
        _nState               := 900;
      END_IF
    END_IF

  100:
    _ipNciChannel.pNciChannelRef^.PlcToNc.MFuncGranted := 0;
    _eCmdActive               := eCmd + e_Ctrl_NciCommand.CMD_DONE;
    _eCmdExec                 := e_Ctrl_NciCommand.CMD_DONE;
END_CASE
CASE _nState OF
  900:
    _eCmdActive               := eCmd + e_Ctrl_NciCommand.CMD_ERROR;
    _eCmdExec                 := e_Ctrl_NciCommand.CMD_ERROR;
END_CASE
END_ACTION

ACTION Channel_Confirm:
CASE _nState OF
  0:
    _hr                       := S_FALSE;
    _nState                   := 10;
END_CASE
CASE _nState OF
  10:
    _eCmdActive               := eCmd + e_Ctrl_NciCommand.CMD_BUSY;
    _eCmdExec                 := e_Ctrl_NciCommand.CMD_BUSY;

    IF (_stMFuncCyclic.HskMFuncReq > 0)
    THEN
      _hr                     := _ipNciChannel.ConfirmHSK(FALSE);
      _nState                 := 20;
    END_IF
END_CASE
CASE _nState OF
  20:
    _hr                       := _ipNciChannel.ConfirmHSK(TRUE);

    IF (_hr = S_OK)
    THEN
      _hr                     := _ipNciChannel.ConfirmHSK(FALSE);
      _nState                 := 100;
    ELSE
      IF (_hr > S_FALSE)
      THEN
        _hr                   := _ipNciChannel.ConfirmHSK(FALSE);
        _nState               := 900;
      END_IF
    END_IF
END_CASE
CASE _nState OF
  100:
    _eCmdActive               := eCmd + e_Ctrl_NciCommand.CMD_DONE;
    _eCmdExec                 := e_Ctrl_NciCommand.CMD_DONE;
END_CASE
CASE _nState OF
  900:
    _eCmdActive               := eCmd + e_Ctrl_NciCommand.CMD_ERROR;
    _eCmdExec                 := e_Ctrl_NciCommand.CMD_ERROR;
END_CASE
END_ACTION

ACTION Channel_LoadProg:
CASE _nState OF
  0:
    _ipNciChannel.pNciChannelRef^.PlcToNc.MFuncGranted := 1;
    _hr                 := S_FALSE;
    _nState              := 10;

  10:
    _ipNciChannel.pNciChannelRef^.PlcToNc.MFuncGranted := 0;
    _eCmdActive          := eCmd + e_Ctrl_NciCommand.CMD_BUSY;
    _eCmdExec            := e_Ctrl_NciCommand.CMD_BUSY;

    IF NOT (len(NcProg) > 10)
    THEN
      _nState             := 900;
    ELSE
      _ipNciChannel.Prog  := NcProg;
  
      _hr                 := _ipNciChannel.LoadProg(FALSE);
  
      _nState             := 20;
    END_IF

  20:
    _ipNciChannel.pNciChannelRef^.PlcToNc.MFuncGranted := 1;
    _hr                 := _ipNciChannel.LoadProg(TRUE);

    IF (_hr = S_OK)
    THEN
      _hr               := _ipNciChannel.LoadProg(FALSE);

      _nState            := 100;
    ELSE
      IF (_hr > S_FALSE)
      THEN
        _hr             := _ipNciChannel.LoadProg(FALSE);

        _nState          := 900;
      END_IF
    END_IF

  100:
    _ipNciChannel.pNciChannelRef^.PlcToNc.MFuncGranted := 0;
    _eCmdActive          := eCmd + e_Ctrl_NciCommand.CMD_DONE;
    _eCmdExec            := e_Ctrl_NciCommand.CMD_DONE;
END_CASE
CASE _nState OF
  900:
    _eCmdActive          := eCmd + e_Ctrl_NciCommand.CMD_ERROR;
    _eCmdExec            := e_Ctrl_NciCommand.CMD_ERROR;
END_CASE
END_ACTION

ACTION Channel_R_Read:
CASE _nState OF
  0:
    _hr           := S_FALSE;
    _nState        := 10;
END_CASE
CASE _nState OF
  10:
    _eCmdActive    := eCmd + e_Ctrl_NciCommand.CMD_BUSY;
    _eCmdExec      := e_Ctrl_NciCommand.CMD_BUSY;

    _iri          := _iRParamIndex;
    _irc          := _iRParamCount;
    _hr           := _ipNciChannel.ReadRParams(FALSE,
                                               ADR(_rRParamsRead),
                                               _iri,
                                               _irc);
    _nState := 20;
END_CASE
CASE _nState OF
  20:
    _hr           := _ipNciChannel.ReadRParams(TRUE,
                                               ADR(_rRParamsRead),
                                               _iri,
                                               _irc);

    IF (_hr = S_OK)
    THEN
      _ipNciChannel.ReadRParams(FALSE,
                                ADR(_rRParamsRead),
                                _iri,
                                _irc);
      _nState      := 100;
    ELSE
      IF (_hr > S_FALSE)
      THEN
        _ipNciChannel.ReadRParams(FALSE,
                                  ADR(_rRParamsRead),
                                  _iri,
                                  _irc);
        _nState    := 900;
      END_IF
    END_IF
END_CASE
CASE _nState OF
  100:
    _eCmdActive    := eCmd + e_Ctrl_NciCommand.CMD_DONE;
    _eCmdExec      := e_Ctrl_NciCommand.CMD_DONE;
END_CASE
CASE _nState OF
  900:
    _eCmdActive    := eCmd + e_Ctrl_NciCommand.CMD_ERROR;
    _eCmdExec      := e_Ctrl_NciCommand.CMD_ERROR;
END_CASE
END_ACTION

ACTION Channel_R_Write:
CASE _nState OF
  0:
    _hr           := S_FALSE;
    _nState        := 10;
END_CASE
CASE _nState OF
  10:
    _eCmdActive    := eCmd + e_Ctrl_NciCommand.CMD_BUSY;
    _eCmdExec      := e_Ctrl_NciCommand.CMD_BUSY;

    _iri          := _iRParamIndex;
    _irc          := _iRParamCount;
    _hr           := _ipNciChannel.WriteRParams(FALSE,
                                                ADR(_rRParamsWrite),
                                                _iri,
                                                _irc);
    _nState := 20;
END_CASE
CASE _nState OF
  20:
    _hr           := _ipNciChannel.WriteRParams(TRUE,
                                                ADR(_rRParamsWrite),
                                                _iri,
                                                _irc);

    IF (_hr = S_OK)
    THEN
      _ipNciChannel.WriteRParams(FALSE,
                                 ADR(_rRParamsWrite),
                                 _iri,
                                 _irc);
      _nState      := 100;
    ELSE
      IF (_hr > S_FALSE)
      THEN
        _ipNciChannel.WriteRParams(FALSE,
                                   ADR(_rRParamsWrite),
                                   _iri,
                                   _irc);
        _nState    := 900;
      END_IF
    END_IF
END_CASE
CASE _nState OF
  100:
    _eCmdActive    := eCmd + e_Ctrl_NciCommand.CMD_DONE;
    _eCmdExec      := e_Ctrl_NciCommand.CMD_DONE;
END_CASE
CASE _nState OF
  900:
    _eCmdActive    := eCmd + e_Ctrl_NciCommand.CMD_ERROR;
    _eCmdExec      := e_Ctrl_NciCommand.CMD_ERROR;
END_CASE
END_ACTION

ACTION Channel_Reset:
CASE _nState OF
  0:
    _hr           := S_FALSE;
    _nState        := 10;
END_CASE
CASE _nState OF
  10:
    _eCmdActive    := eCmd + e_Ctrl_NciCommand.CMD_BUSY;
    _eCmdExec      := e_Ctrl_NciCommand.CMD_BUSY;

    _hr           := _ipNciChannel.ItpReset(FALSE);

    _nState := 20;
END_CASE
CASE _nState OF
  20:
    _hr           := _ipNciChannel.ItpReset(TRUE);

    IF (_hr = S_OK)
    THEN
      _ipNciChannel.ItpReset(FALSE);
      _nState      := 100;
    ELSE
      IF (_hr > S_FALSE)
      THEN
        _ipNciChannel.ItpReset(FALSE);
        _nState    := 900;
      END_IF
    END_IF
END_CASE
CASE _nState OF
  100:
    _eCmdActive    := eCmd + e_Ctrl_NciCommand.CMD_DONE;
    _eCmdExec      := e_Ctrl_NciCommand.CMD_DONE;
END_CASE
CASE _nState OF
  900:
    _eCmdActive    := eCmd + e_Ctrl_NciCommand.CMD_ERROR;
    _eCmdExec      := e_Ctrl_NciCommand.CMD_ERROR;
END_CASE
END_ACTION

ACTION Channel_Restart:
CASE _nState OF
  0:
    _hr                     := S_FALSE;
    _nState                  := 10;
END_CASE
CASE _nState OF
  10:
    _eCmdActive              := eCmd + e_Ctrl_NciCommand.CMD_BUSY;
    _eCmdExec                := e_Ctrl_NciCommand.CMD_BUSY;

    _hr                     := _ipNciChannel.StepOnAfterEStop(FALSE);

    _nState                  := 20;
END_CASE
CASE _nState OF
  20:
    _hr                     := _ipNciChannel.StepOnAfterEStop(TRUE);

    IF (_hr = S_OK)
    THEN
      _hr                   := _ipNciChannel.StepOnAfterEStop(FALSE);
      _nState                := 100;
    ELSE
      IF (_hr > S_FALSE)
      THEN
        _hr                 := _ipNciChannel.StepOnAfterEStop(FALSE);
        _nState              := 900;
      END_IF
    END_IF
END_CASE
CASE _nState OF
  100:
    _eCmdActive              := eCmd + e_Ctrl_NciCommand.CMD_DONE;
    _eCmdExec                := e_Ctrl_NciCommand.CMD_DONE;
END_CASE
CASE _nState OF
  900:
    _eCmdActive              := eCmd + e_Ctrl_NciCommand.CMD_ERROR;
    _eCmdExec                := e_Ctrl_NciCommand.CMD_ERROR;
END_CASE
END_ACTION

ACTION Channel_Start:
CASE _nState OF
  0:
    _hr                     := S_FALSE;
    _nState                  := 10;
END_CASE
CASE _nState OF
  10:
    _eCmdActive              := eCmd + e_Ctrl_NciCommand.CMD_BUSY;
    _eCmdExec                := e_Ctrl_NciCommand.CMD_BUSY;

    _hr                     := _ipNciChannel.StartStop(FALSE, FALSE);

    _nState                  := 20;
END_CASE
CASE _nState OF
  20:
    _hr                     := _ipNciChannel.StartStop(TRUE, FALSE);

    IF (_hr = S_OK)
    THEN
      _hr                   := _ipNciChannel.StartStop(FALSE, FALSE);
      _nState                := 100;
    ELSE
      IF (_hr > S_FALSE)
      THEN
        _hr                 := _ipNciChannel.StartStop(FALSE, FALSE);
        _nState              := 900;
      END_IF
    END_IF
END_CASE
CASE _nState OF
  100:
    _eCmdActive              := eCmd + e_Ctrl_NciCommand.CMD_DONE;
    _eCmdExec                := e_Ctrl_NciCommand.CMD_DONE;
END_CASE
CASE _nState OF
  900:
    _eCmdActive              := eCmd + e_Ctrl_NciCommand.CMD_ERROR;
    _eCmdExec                := e_Ctrl_NciCommand.CMD_ERROR;
END_CASE
END_ACTION

ACTION Channel_Stop:
CASE _nState OF
  0:
    _hr                     := S_FALSE;
    _nState                  := 10;
END_CASE
CASE _nState OF
  10:
    _eCmdActive              := eCmd + e_Ctrl_NciCommand.CMD_BUSY;
    _eCmdExec                := e_Ctrl_NciCommand.CMD_BUSY;

    _hr                     := _ipNciChannel.StartStop(FALSE, FALSE);

    _nState                  := 20;
END_CASE
CASE _nState OF
  20:
    _hr                     := _ipNciChannel.StartStop(FALSE, TRUE);

    IF (_hr = S_OK)
    THEN
      _hr                   := _ipNciChannel.StartStop(FALSE, FALSE);
      _nState                := 100;
    ELSE
      IF (_hr > S_FALSE)
      THEN
        _hr                 := _ipNciChannel.StartStop(FALSE, FALSE);
        _nState              := 900;
      END_IF
    END_IF
END_CASE
CASE _nState OF
  100:
    _eCmdActive              := eCmd + e_Ctrl_NciCommand.CMD_DONE;
    _eCmdExec                := e_Ctrl_NciCommand.CMD_DONE;
END_CASE
CASE _nState OF
  900:
    _eCmdActive              := eCmd + e_Ctrl_NciCommand.CMD_ERROR;
    _eCmdExec                := e_Ctrl_NciCommand.CMD_ERROR;
END_CASE
END_ACTION

PROPERTY ChnId : udint
GET
ChnId := _ipNciChannel.pNciChannelRef^.NcToPlc.ChnId;
END_GET
END_PROPERTY

METHOD Cycle
VAR_INPUT
END_VAR
// call NCI
_fbNciChannel();
_ipNciChannel := _fbNciChannel;


// cyclic plausibility checks
IF Init() <> S_OK 
THEN
  eState  := e_Ctrl_NciCommand.NO_INIT;
  RETURN;
END_IF


// cyclic data for M func from NCI interface
_stMFuncCyclic.FastMFuncMask  := _ipNciChannel.pNciChannelRef^.NcToPlc.FastMFuncMask;
_stMFuncCyclic.HskMFuncNo     := _ipNciChannel.pNciChannelRef^.NcToPlc.HskMFuncNo;
_stMFuncCyclic.HskMFuncReq    := _ipNciChannel.pNciChannelRef^.NcToPlc.HskMFuncReq;
_stMFuncCyclic.HFuncValue     := _ipNciChannel.pNciChannelRef^.NcToPlc.HFuncValue;

// M-Func to catch
IF _ipNciChannel.HSK 
THEN
  _nMFunc := _ipNciChannel.MFunc;
END_IF


// cmd change
IF (_eCmd <> _eCmdOld) OR
   (_eCmd = 0)
THEN
  _eCmdState                  := _eCmd;
  _nState      := _nStateSS1  := 0;
  _nMFunc                     := 0;
  _stMsg.sText                := '';
  _sState                     := '';
END_IF


CASE _eCmdState OF

  e_Ctrl_NciCommand.INIT:
    _eCmdActive                := _eCmdState + e_Ctrl_NciCommand.CMD_DONE;
    _eCmdExec                  := e_Ctrl_NciCommand.CMD_DONE;
    _nState                    := 0;

  e_Ctrl_NciCommand.IDLE:
    _eCmdActive                := _eCmdState + e_Ctrl_NciCommand.CMD_BUSY;
    _eCmdExec                  := e_Ctrl_NciCommand.CMD_BUSY;

    _uiStateItp                := _ipNciChannel.GetItpState();

    IF (_uiStateItp = TO_UINT(E_NCI_INTERPRETER_STATE.NCI_INTERPRETER_IDLE)) OR
       (_uiStateItp = TO_UINT(E_NCI_INTERPRETER_STATE.NCI_INTERPRETER_READY))
    THEN
      _eCmdActive              := _eCmdState + e_Ctrl_NciCommand.CMD_DONE;
      _eCmdExec                := e_Ctrl_NciCommand.CMD_DONE;
      _nState                  := 0;
    END_IF


  e_Ctrl_NciCommand.RESET:
    // reset for error
    // after reset nc file has to be loaded again
    Channel_Reset();

  e_Ctrl_NciCommand.LOAD_PROG:
    // set property NcProg before use
    // load nc file
    // syntax check on load done by NCI
    // error case: syntax check failed
    Channel_LoadProg();

  e_Ctrl_NciCommand.BUILD_GROUP:
    // set property GroupAxisConfig before use
    Channel_BuildGroup();

  e_Ctrl_NciCommand.CLEAR_GROUP:
    Channel_ClearGroup();

  e_Ctrl_NciCommand.START:
    // starts nc file execution
    Channel_Start();

  e_Ctrl_NciCommand.STOP,
  e_Ctrl_NciCommand.STO_STOP:
    Channel_Stop();

  e_Ctrl_NciCommand.RESTART_STEP_ON:
    // sart from last nc block
    Channel_Restart();

  e_Ctrl_NciCommand.M_FUNC_QUIT:
    Channel_Confirm();

  e_Ctrl_NciCommand.READ_R_PARA:
    Channel_R_Read();

  e_Ctrl_NciCommand.WRITE_R_PARA:
    Channel_R_Write();

  ELSE
    _eState                  := e_Ctrl_NciCommand.NO_INIT;
    _sState                  := concat(TO_STRING(_eCmdState), ' NOT valid eCmd');
    RETURN;
END_CASE

_eState                      := _eCmdActive;
_sState                      := TO_STRING(_eCmdState);
_sCmd                        := TO_STRING(eCmd);
_sCmdExec                    := TO_STRING(_eCmdExec);


IF (_eCmdOld <> eCmd)
THEN
  _sCmdOld                   := TO_STRING(_eCmdOld);
  _stMsg.eType               := E_MessageType.eMessageInfo;
  _stMsg.eDevice             := E_Device.NciChannelCtrl + TO_DINT(ChnId);
  _stMsg.eSubdevice          := e_Subdevice.Ctrl_Nci_Cmd;
  _stMsg.iErrorNumber        := _nChnId;

  _stMsg.sText               := 'change ';
  _stMsg.sText               := Tc2_Standard.CONCAT(_stMsg.sText, _sCmdOld);
  _stMsg.sText               := Tc2_Standard.CONCAT(_stMsg.sText, ' to ');
  _stMsg.sText               := Tc2_Standard.CONCAT(_stMsg.sText, sCmd);
  f_MessageSet(_stMsg);
END_IF

IF (_eCmdExecOld <> _eCmdExec)
THEN
  _stMsg.eType               := E_MessageType.eMessageInfo;
  _stMsg.eDevice             := E_Device.NciChannelCtrl + TO_DINT(ChnId);
  _stMsg.eSubdevice          := e_Subdevice.Ctrl_Nci_Cmd;
  _stMsg.iErrorNumber        := _nChnId;

  _stMsg.sText               := Tc2_Standard.CONCAT(sCmd, ' function: ');
  _stMsg.sText               := Tc2_Standard.CONCAT(_stMsg.sText, TO_STRING(_eCmdExec));
  f_MessageSet(_stMsg);
END_IF

_eCmdOld                     := eCmd;
_eCmdExecOld                 := _eCmdExec;
END_METHOD

PROPERTY eCmd : e_Ctrl_NciCommand
GET
eCmd := _eCmd;
END_GET
SET
_eCmd := eCmd;
END_SET
END_PROPERTY

PROPERTY eState : e_Ctrl_NciCommand
GET
eState := _eState;
END_GET
SET
_eState := eState;
END_SET
END_PROPERTY

PROPERTY GroupAxisConfig : ST_3D_Group
GET
VAR
  st3DGroup       : ST_3D_Group;
  stNciExt3dGroup : NCI_EXT3DGROUP;
END_VAR
stNciExt3dGroup := _fbNciChannel.ItpAxes;
memcpy(ADR(st3DGroup), ADR(stNciExt3dGroup), SIZEOF(st3DGroup));
GroupAxisConfig := st3DGroup;
END_GET
SET
VAR
  st3DGroup       : ST_3D_Group;
  stNciExt3dGroup : NCI_EXT3DGROUP;
END_VAR
st3DGroup := GroupAxisConfig;
memcpy(ADR(stNciExt3dGroup), ADR(st3DGroup), SIZEOF(stNciExt3dGroup));

_fbNciChannel.CfgAxes := stNciExt3dGroup;
END_SET
END_PROPERTY

PROPERTY I_AuxAxis : array[1..GVL_NCI.cAuxAxisCount] of I_McAxis
GET
I_AuxAxis := THIS^._ipAuxAxis;
END_GET
SET
VAR
  idx : DINT;
END_VAR
THIS^._ipAuxAxis := I_AuxAxis;

_iAuxCountConfigured := 0;
FOR idx := 1 TO GVL_NCI.cAuxAxisCount
DO
  IF (_ipAuxAxis[idx] <> 0)
  THEN
    _iAuxCountConfigured := _iAuxCountConfigured + 1;
  END_IF
END_FOR
END_SET
END_PROPERTY

PROPERTY I_McAxis : array[1..GVL_NCI.cMcAxisCount] of I_McAxis
GET
I_McAxis := THIS^._ipMcsAxis;
END_GET
SET
VAR
  idx : DINT;
END_VAR
_ipMcsAxis := I_McAxis;

_iMcCountConfigured := 0;
FOR idx := 1 TO GVL_NCI.cMcAxisCount
DO
  IF (_ipMcsAxis[idx] <> 0)
  THEN
    _iMcCountConfigured := _iMcCountConfigured + 1;
  END_IF
END_FOR
END_SET
END_PROPERTY

PROPERTY I_NcChannel : I_NciChannel
GET
I_NcChannel := _fbNciChannel;
END_GET
END_PROPERTY

METHOD PRIVATE Init : HRESULT
VAR_INST
  hr    : HRESULT   := S_FALSE;
END_VAR
IF hr <> S_OK 
THEN

  _nChnId := _fbNciChannel.pNciChannelRef^.NcToPlc.ChnId;
  IF (_nChnId = 0)
  THEN
    _sState    := 'CannelId = 0';
    Init      := hr := -1;
    RETURN;
  ELSE
    _sState    := concat('CannelId = ', TO_STRING(_nChnId));
  END_IF
  
  _iMcCount   := 0;
  _iAuxCount  := 0;
  
  FOR _mdx := 1 TO GVL_NCI.cMcAxisCount
  DO
    IF (_ipMcsAxis[_mdx] <> 0)
    THEN
      _iMcCount := _iMcCount + 1;
    END_IF
  END_FOR
  
  FOR _adx := 1 TO GVL_NCI.cAuxAxisCount
  DO
    IF (_ipAuxAxis[_adx] <> 0)
    THEN
      _iAuxCount := _iAuxCount + 1;
    END_IF
  END_FOR
  
  IF (_iAuxCount <> _iAuxCountConfigured) OR
     (_iMcCount  <> _iMcCountConfigured) 
  THEN
    _sState                    := 'Axis count mismatch';

    // get first occurance of error
    IF NOT _bMcAxisMismatch
    THEN
      _stMsg.eType             := E_MessageType.eMessageError;
      _stMsg.eDevice           := _ChannelDevice;
      _stMsg.eSubdevice        := e_Subdevice.General;
      _stMsg.iErrorNumber      := e_NciChannelError.e_AxisConfigurationMismatch_McAxis;
      _stMsg.sText             := 'MC Axis count mismatch';
      f_MessageSet(_stMsg);
    END_IF
  
    // get first ocurrance of error
    IF NOT _bAuxAxisMismatch
    THEN
      _stMsg.eType             := E_MessageType.eMessageError;
      _stMsg.eDevice           := _ChannelDevice;
      _stMsg.eSubdevice        := e_Subdevice.General;
      _stMsg.iErrorNumber      := e_NciChannelError.e_AxisConfigurationMismatch_AuxAxis;
      _stMsg.sText             := 'Aux Axis count mismatch';
      f_MessageSet(_stMsg);
    END_IF
  ELSE
    // get change of error
    IF _bMcAxisMismatch
    THEN
      _stMsg.eType             := E_MessageType.eMessageInfo;
      _stMsg.eDevice           := _ChannelDevice;
      _stMsg.eSubdevice        := e_Subdevice.General;
      _stMsg.iErrorNumber      := e_NciChannelError.e_AxisConfigurationMismatch_McAxis;
      _stMsg.sText             := 'MC Axis count match';
      f_MessageSet(_stMsg);
    END_IF
  
    // get change of error
    IF _bAuxAxisMismatch
    THEN
      _stMsg.eType             := E_MessageType.eMessageInfo;
      _stMsg.eDevice           := _ChannelDevice;
      _stMsg.eSubdevice        := e_Subdevice.General;
      _stMsg.iErrorNumber      := e_NciChannelError.e_AxisConfigurationMismatch_AuxAxis;
      _stMsg.sText             := 'Aux Axis count match';
      f_MessageSet(_stMsg);
    END_IF
  END_IF
  
  _bMcAxisMismatch  := (_iMcCount  <> _iMcCountConfigured);
  _bAuxAxisMismatch := (_iAuxCount <> _iAuxCountConfigured);
  
  IF (_bMcAxisMismatch) OR
     (_bAuxAxisMismatch)
  THEN
    _nErrorId    := SEL(_bMcAxisMismatch, _nErrorId, (_nErrorId OR 2#0001));
    _nErrorId    := SEL(_bAuxAxisMismatch,_nErrorId, (_nErrorId OR 2#001));
    _bError      := TRUE;
    RETURN;
  END_IF 


  _bError                  := FALSE;
  hr                       := S_OK;
  _eCmdState               := e_Ctrl_NciCommand.INIT;
  // initial assignement, 
  // if required; change on calling BuildGroup
  _fbNciChannel.I_AuxAxis := I_AuxAxis;
  _fbNciChannel.I_McAxis  := I_McAxis;
END_IF

//Return Value
Init := hr;
END_METHOD

PROPERTY M_FuncReq : word
GET
M_FuncReq := _fbNciChannel.pNciChannelRef^.NcToPlc.HskMFuncReq;
END_GET
END_PROPERTY

PROPERTY NcProg : string(255)
GET
NcProg := _sProg;
END_GET
SET
_sProg := NcProg;
END_SET
END_PROPERTY

PROPERTY R_Param_Read : ARRAY [0..GVL_NCI.cRParamCount] OF lreal
GET
R_Param_Read := _rRParamsRead;
END_GET
SET
_rRParamsRead := R_Param_Read;
END_SET
END_PROPERTY

PROPERTY R_Param_Write : ARRAY [0..GVL_NCI.cRParamCount] OF lreal
GET
R_Param_Write := _rRParamsWrite;
END_GET
SET
_rRParamsWrite := R_Param_Write;
END_SET
END_PROPERTY

PROPERTY R_ParamCount : DINT
GET
R_ParamCount := _iRParamCount;
END_GET
SET
_iRParamCount := R_ParamCount;
END_SET
END_PROPERTY

PROPERTY R_ParamIndex : DINT
GET
R_ParamIndex := _iRParamIndex;
END_GET
SET
_iRParamIndex := R_ParamIndex;
END_SET
END_PROPERTY

PROPERTY sCmd : string
GET
sCmd := _sCmd;
END_GET
SET
_sCmd := sCmd;
END_SET
END_PROPERTY

END_FUNCTION_BLOCK

// ---- POUs/NCI/FB_NciChannel.TcPOU
FUNCTION_BLOCK FB_NciChannel IMPLEMENTS I_NciChannel
VAR
  stMsg                 : ST_Message;
  ChannelDevice         : e_Device;

//MCS-Axes
  _ipMcsAxis            : ARRAY[1..GVL_NCI.cMcAxisCount] OF I_McAxis;
  _iMcCount,
  _iMcCountConfigured   : DINT;
  _bMcAxisMismatch      : BOOL;

//Aux-Axes
  _ipAuxAxis            : ARRAY[1..GVL_NCI.cAuxAxisCount] OF I_McAxis;
  _iAuxCount,
  _iAuxCountConfigured  : DINT;
  _bAuxAxisMismatch     : BOOL;

  _bErrorCyclicChecks   : BOOL;


//NCI-Channel reference
  _refNciChannelRef     : ST_NciChannel_Ref;

//NCI-Error
  _ErrorCode            : UDINT;
  
//NCI-Group
  fbBuildGroup          : Tc2_NCI.CfgBuildExt3DGroup;
  fbClearGroup          : Tc2_NCI.CfgReconfigGroup;

  _stCfgAxes            : Tc2_NCI.NCI_EXT3DGROUP;   //Configured Group Axes

  _fOverride            : LREAL := 100;

  _Build, 
  _Move                 : BOOL;

  _mdx,
  _adx                  : UINT;
  
//NCI-Program
  fbLoadProg            : Tc2_NCI.ItpLoadProgEx;

  _sProg                : STRING(255);

//Interpreter
  fbReset               : Tc2_NCI.ItpResetEx2;
  fbStartStop           : Tc2_NCI.ItpStartStopEx;
  fbEStop               : Tc2_NCI.ItpEStopEx;
  fbStepOnAfterEStop    : Tc2_NCI.ItpStepOnAfterEStopEx;

  fbItpConfirmHsk       : Tc2_NCI.ItpConfirmHsk;
  fbItpReadRParams      : Tc2_NCI.ItpReadRParamsEx;
  fbItpWriteRParams     : Tc2_NCI.ItpWriteRParamsEx;
  fbItpDelDtg           : Tc2_NCI.ItpDelDtgEx;

  
//ADS-Communication
  fbReadLine            : Tc2_System.ADSREADEX;

END_VAR

IF NOT (_refNciChannelRef.NcToPlc.ChnId <> 0)
THEN
  RETURN;
END_IF

ChannelDevice := e_Device.NciChannel + (_refNciChannelRef.NcToPlc.ChnId);

_iMcCount   := 0;
_iAuxCount  := 0;

FOR _mdx := 1 TO GVL_NCI.cMcAxisCount
DO
  IF (_ipMcsAxis[_mdx] <> 0)
  THEN
    _iMcCount := _iMcCount + 1;
  END_IF
END_FOR

FOR _adx := 1 TO GVL_NCI.cAuxAxisCount
DO
  IF (_ipAuxAxis[_adx] <> 0)
  THEN
    _iAuxCount := _iAuxCount + 1;
  END_IF
END_FOR

IF (_iAuxCount <> _iAuxCountConfigured) OR
   (_iMcCount  <> _iMcCountConfigured) 
THEN
  // get first occurance of error
  IF NOT _bMcAxisMismatch
  THEN
    stMsg.eType             := E_MessageType.eMessageError;
    stMsg.eDevice           := ChannelDevice;
    stMsg.eSubdevice        := e_Subdevice.General;
    stMsg.iErrorNumber      := e_NciChannelError.e_AxisConfigurationMismatch_McAxis;
    stMsg.sText             := 'MC Axis count mismatch';
    f_MessageSet(stMsg);
  END_IF

  // get first ocurrance of error
  IF NOT _bAuxAxisMismatch
  THEN
    stMsg.eType             := E_MessageType.eMessageError;
    stMsg.eDevice           := ChannelDevice;
    stMsg.eSubdevice        := e_Subdevice.General;
    stMsg.iErrorNumber      := e_NciChannelError.e_AxisConfigurationMismatch_AuxAxis;
    stMsg.sText             := 'Aux Axis count mismatch';
    f_MessageSet(stMsg);
  END_IF
ELSE
  // get change of error
  IF _bMcAxisMismatch
  THEN
    stMsg.eType             := E_MessageType.eMessageInfo;
    stMsg.eDevice           := ChannelDevice;
    stMsg.eSubdevice        := e_Subdevice.General;
    stMsg.iErrorNumber      := e_NciChannelError.e_AxisConfigurationMismatch_McAxis;
    stMsg.sText             := 'MC Axis count match';
    f_MessageSet(stMsg);
  END_IF

  // get change of error
  IF _bAuxAxisMismatch
  THEN
    stMsg.eType             := E_MessageType.eMessageInfo;
    stMsg.eDevice           := ChannelDevice;
    stMsg.eSubdevice        := e_Subdevice.General;
    stMsg.iErrorNumber      := e_NciChannelError.e_AxisConfigurationMismatch_AuxAxis;
    stMsg.sText             := 'Aux Axis count match';
    f_MessageSet(stMsg);
  END_IF
END_IF

_bMcAxisMismatch  := (_iMcCount  <> _iMcCountConfigured);
_bAuxAxisMismatch := (_iAuxCount <> _iAuxCountConfigured);

(*
===============================================================
Implementation of Tc2_NCI.CfgBuildExt3DGroup

  Builds complete NCI-Group with all configured axes
===============================================================
*)
METHOD BuildGroup : HRESULT
VAR_INPUT
  Execute        : BOOL;
END_VAR
VAR_INST
  istate          : DINT;
  stMsg           : ST_Message;
  hr              : HRESULT;
END_VAR


IF NOT Execute
THEN
  istate := 0;
END_IF


CASE istate OF
  0:
    hr:= S_FALSE;
    fbBuildGroup( bExecute  := FALSE, 
                  nGroupId  := ItpGetGroupId(sNciToPlc:=_refNciChannelRef.NcToPlc) , 
                  nXAxisId  := _stCfgAxes.nXAxisId,
                  nYAxisId  := _stCfgAxes.nYAxisId, 
                  nZAxisId  := _stCfgAxes.nZAxisId, 
                  nQ1AxisId := _stCfgAxes.nQ1AxisId,
                  nQ2AxisId := _stCfgAxes.nQ2AxisId, 
                  nQ3AxisId := _stCfgAxes.nQ3AxisId, 
                  nQ4AxisId := _stCfgAxes.nQ4AxisId, 
                  nQ5AxisId := _stCfgAxes.nQ5AxisId);

    IF Execute
    THEN
      istate                := 10;
    END_IF
END_CASE
CASE istate OF
  10:
    fbBuildGroup( bExecute  := TRUE, 
                  nGroupId  := ItpGetGroupId(sNciToPlc:=_refNciChannelRef.NcToPlc));

    IF fbBuildGroup.bBusy 
    THEN
      hr:= S_FALSE;
    
    ELSIF fbBuildGroup.bErr 
    THEN
      istate                := 99;

      stMsg.eType           := E_MessageType.eMessageError;
      stMsg.eDevice         := ChannelDevice;
      stMsg.eSubdevice      := e_Subdevice.fbBuildGroup;
      stMsg.iErrorNumber    := fbBuildGroup.nErrId;
      stMsg.sText           := concat('BuildGroup Error: ', TO_STRING(fbBuildGroup.nErrId));
      f_MessageSet(stMsg);

      hr:= TO_DINT(fbBuildGroup.nErrId);

    ELSE
      istate                := 100;

      stMsg.eType           := E_MessageType.eMessageInfo;
      stMsg.eDevice         := ChannelDevice;
      stMsg.eSubdevice      := e_Subdevice.fbBuildGroup;
      stMsg.iErrorNumber    := fbBuildGroup.nErrId;
      stMsg.sText           := concat('BuildGroup Done: ', TO_STRING(fbBuildGroup.nErrId));
      f_MessageSet(stMsg);
    END_IF
END_CASE
CASE istate OF
  100:
    hr:= S_OK;
END_CASE

//Return Result
BuildGroup:= hr;
END_METHOD

(*
===============================================================
NCI-Group configured axes structure
===============================================================
*)
PROPERTY CfgAxes : Tc2_NCI.NCI_EXT3DGROUP
SET
_stCfgAxes := CfgAxes;  //Configured Group Axes
END_SET
END_PROPERTY

(*
===============================================================
Implementation of Tc2_NCI.CfgReconfigGroup

  remove all axes from NCI-Group
===============================================================
*)
METHOD ClearGroup : HRESULT
VAR_INPUT
  Execute   : BOOL;
END_VAR
VAR_INST
  istate    : DINT;
  stMsg     : ST_Message;
  hr        : HRESULT;
END_VAR

IF NOT Execute
THEN
  istate := 0;
END_IF


CASE istate OF
  0:
    hr:= S_FALSE;
    fbClearGroup( bExecute:= FALSE, 
                  nGroupId:= ItpGetGroupId(sNciToPlc:= _refNciChannelRef.NcToPlc));

    IF Execute
    THEN
      istate                := 10;
    END_IF
END_CASE
CASE istate OF
  10:
    fbClearGroup( bExecute:= TRUE, 
                  nGroupId:= ItpGetGroupId(sNciToPlc:= _refNciChannelRef.NcToPlc));

    IF fbClearGroup.bBusy 
    THEN
      hr:= S_FALSE;
    
    ELSIF fbClearGroup.bErr 
    THEN
      istate                := 99;

      stMsg.eType           := E_MessageType.eMessageError;
      stMsg.eDevice         := ChannelDevice;
      stMsg.eSubdevice      := e_Subdevice.fbClearGroup;
      stMsg.iErrorNumber    := fbClearGroup.nErrId;
      stMsg.sText           := concat('BuildGroup Error: ', TO_STRING(fbClearGroup.nErrId));
      f_MessageSet(stMsg);

      hr:= TO_DINT(fbClearGroup.nErrId);

    ELSE
      istate                := 100;

      stMsg.eType           := E_MessageType.eMessageInfo;
      stMsg.eDevice         := ChannelDevice;
      stMsg.eSubdevice      := e_Subdevice.fbClearGroup;
      stMsg.iErrorNumber    := fbClearGroup.nErrId;
      stMsg.sText           := concat('ClearGroup Done: ', TO_STRING(fbClearGroup.nErrId));
      f_MessageSet(stMsg);

    END_IF
END_CASE
CASE istate OF
  100:
    hr := S_OK;
END_CASE

//Return Result
ClearGroup:= hr;
END_METHOD

(*
===============================================================
Implementation of Tc2_NCI.ItpConfirmHsk

  acknowledge M-Function
===============================================================
*)
METHOD ConfirmHSK : HRESULT
VAR_INPUT
  Execute   : BOOL;
END_VAR
VAR_INST
  hr        : HRESULT;
  istate    : DINT;
  stMsg     : ST_Message;
END_VAR

IF NOT Execute
THEN
  istate              := 0;
END_IF


CASE istate OF
  0:
    hr                                        := S_FALSE;
    _refNciChannelRef.PlcToNc.MFuncGranted    := 0;

    IF Execute
    THEN
      IF (_refNciChannelRef.PlcToNc.ChnAxesOvr > 0) AND NOT
         (_refNciChannelRef.NcToPlc.ChnState.8)
      THEN
        IF (_refNciChannelRef.NcToPlc.HskMFuncReq = 1)
        THEN
          istate                              := 10;
        END_IF
      END_IF
    END_IF

  10:
    _refNciChannelRef.PlcToNc.MFuncGranted    := 1;

    IF (_refNciChannelRef.NcToPlc.HskMFuncReq = 0)
    THEN
      istate                                  := 100;
      _refNciChannelRef.PlcToNc.MFuncGranted  := 0;
    END_IF
END_CASE
CASE istate OF
  100:
    hr                                        := S_OK;
END_CASE

//Return Result
ConfirmHSK:= hr;
END_METHOD

// delete distance to go
METHOD DelDTG : HRESULT
VAR_INPUT
  Execute     : BOOL;
END_VAR
VAR_INST
  istate      : DINT;
  stMsg       : ST_Message;
  hr          : HRESULT;
END_VAR

IF NOT Execute
THEN
  istate := 0;
END_IF


CASE istate OF
  0:
    hr:= S_FALSE;

    fbItpDelDtg(sNciToPlc   := _refNciChannelRef.NcToPlc, 
                bExecute    := FALSE);

    IF Execute
    THEN
      istate                := 10;
    END_IF
END_CASE
CASE istate OF
  10:
    fbItpDelDtg(sNciToPlc   := _refNciChannelRef.NcToPlc, 
                bExecute    := TRUE);

    IF fbItpDelDtg.bBusy 
    THEN
      hr:= S_FALSE;
    
    ELSIF fbItpDelDtg.bErr 
    THEN
      istate                := 99;

      stMsg.eType           := E_MessageType.eMessageError;
      stMsg.eDevice         := ChannelDevice;
      stMsg.eSubdevice      := e_Subdevice.fbDelDtgItp;
      stMsg.iErrorNumber    := fbItpDelDtg.nErrId;
      stMsg.sText           := concat('fbItpDelDtg Error: ', TO_STRING(fbItpDelDtg.nErrId));
      f_MessageSet(stMsg);

      hr:= TO_DINT(stMsg.iErrorNumber);

    ELSE
      istate                := 100;

      stMsg.eType           := E_MessageType.eMessageInfo;
      stMsg.eDevice         := ChannelDevice;
      stMsg.eSubdevice      := e_Subdevice.fbDelDtgItp;
      stMsg.iErrorNumber    := fbItpDelDtg.nErrId;
      stMsg.sText           := concat('fbItpDelDtg Done: ', TO_STRING(fbItpDelDtg.nErrId));
      f_MessageSet(stMsg);
    END_IF
END_CASE
CASE istate OF
  100:
    hr:= S_OK;
END_CASE

//Return Result
DelDTG:= hr;
END_METHOD

(*
===============================================================
Error-Flag
===============================================================
*)
PROPERTY Error : BOOL
GET
// get error from channel state
Error:= Error_Get();
END_GET
END_PROPERTY

METHOD Error_Get : BOOL
VAR_INST
  i               : INT;
  stMsg           : ST_Message;
END_VAR
//Return Value
Error_Get:= FALSE;

//NciChannel
IF _refNciChannelRef.NcToPlc.ErrorCode <> 0 
THEN
  stMsg.eType         := E_MessageType.eMessageError;
  stMsg.eDevice       := ChannelDevice;
  stMsg.eSubdevice    := e_Subdevice.Get_Error;
  stMsg.iErrorNumber  := _refNciChannelRef.NcToPlc.ErrorCode;
  stMsg.sText         := concat('NCI-Error: ', TO_STRING(_refNciChannelRef.NcToPlc.ErrorCode));
  f_MessageSet(stMsg);
  Error_Get:= TRUE;
  RETURN;
END_IF
END_METHOD

(*
===============================================================
Implementation of Tc2_NCI.ItpEStopEx
===============================================================
*)
METHOD EStop : HRESULT
VAR_INPUT
  Execute   : BOOL;
END_VAR
VAR_INST
  istate    : DINT;
  stMsg     : ST_Message;
  hr        : HRESULT;
END_VAR

IF NOT Execute
THEN
  istate := 0;
END_IF


CASE istate OF
  0:
    hr                    := S_FALSE;

    fbEStop(sNciToPlc     := _refNciChannelRef.NcToPlc, 
            bExecute      := FALSE);

    IF Execute
    THEN
      istate              := 10;
    END_IF
END_CASE
CASE istate OF
  10:
    fbEStop(sNciToPlc     := _refNciChannelRef.NcToPlc, 
            bExecute      := TRUE);

    IF fbEStop.bBusy 
    THEN
      hr:= S_FALSE;
    
    ELSIF fbEStop.bErr 
    THEN
      istate                := 99;

      stMsg.eType           := E_MessageType.eMessageError;
      stMsg.eDevice         := ChannelDevice;
      stMsg.eSubdevice      := e_Subdevice.fbEStopItp;
      stMsg.iErrorNumber    := fbEStop.nErrId;
      stMsg.sText           := concat('fbEStopItp Error: ', TO_STRING(fbEStop.nErrId));
      f_MessageSet(stMsg);

      hr:= TO_DINT(fbEStop.nErrId);
    ELSE
      istate                := 100;

      stMsg.eType           := E_MessageType.eMessageInfo;
      stMsg.eDevice         := ChannelDevice;
      stMsg.eSubdevice      := e_Subdevice.fbEStopItp;
      stMsg.iErrorNumber    := fbEStop.nErrId;
      stMsg.sText           := concat('fbEStopItp Done: ', TO_STRING(fbEStop.nErrId));
      f_MessageSet(stMsg);
    END_IF
END_CASE
CASE istate OF
  100:
    hr:= S_OK;
END_CASE

//Return Result
EStop:= hr;
END_METHOD

METHOD GetChannelOverride : real
VAR_INPUT
END_VAR
GetChannelOverride := TO_REAL(_refNciChannelRef.PlcToNc.ChnAxesOvr)/10_000.0;
END_METHOD

METHOD GetItpState : uint
VAR_INPUT
END_VAR
GetItpState := _refNciChannelRef.NcToPlc.ItpState;
END_METHOD

(*
===============================================================
Handshake: Announce and acknowledge M-Functions
===============================================================
*)
PROPERTY HSK : BOOL
GET

HSK :=  TO_BOOL(_refNciChannelRef.NcToPlc.HskMFuncReq);
END_GET
END_PROPERTY

PROPERTY I_AuxAxis : ARRAY[1..GVL_NCI.cAuxAxisCount] OF I_McAxis
SET
VAR
  idx : DINT;
END_VAR
_ipAuxAxis := I_AuxAxis;

_iAuxCountConfigured := 0;
FOR idx := 1 TO GVL_NCI.cAuxAxisCount
DO
  IF (_ipAuxAxis[idx] <> 0)
  THEN
    _iAuxCountConfigured := _iAuxCountConfigured + 1;
  END_IF
END_FOR
END_SET
END_PROPERTY

PROPERTY I_McAxis : array[1..GVL_NCI.cMcAxisCount] of I_McAxis
SET
VAR
  idx : dint;
END_VAR
_ipMcsAxis := I_McAxis;

_iMcCountConfigured := 0;
FOR idx := 1 TO GVL_NCI.cMcAxisCount
DO
  IF (_ipMcsAxis[idx] <> 0)
  THEN
    _iMcCountConfigured := _iMcCountConfigured + 1;
  END_IF
END_FOR
END_SET
END_PROPERTY

(*
===============================================================
NCI-Group configured axes structure
===============================================================
*)
PROPERTY ItpAxes : Tc2_NCI.NCI_EXT3DGROUP
GET
VAR
  stItpAxes     :Tc2_NCI.NCI_EXT3DGROUP;
END_VAR

stItpAxes.nXAxisId := _refNciChannelRef.NcToPlc.AcsAxisIDs[0];
stItpAxes.nYAxisId := _refNciChannelRef.NcToPlc.AcsAxisIDs[1];
stItpAxes.nZAxisId := _refNciChannelRef.NcToPlc.AcsAxisIDs[2];
stItpAxes.nQ1AxisId := _refNciChannelRef.NcToPlc.AcsAxisIDs[3];
stItpAxes.nQ2AxisId := _refNciChannelRef.NcToPlc.AcsAxisIDs[4];
stItpAxes.nQ3AxisId := _refNciChannelRef.NcToPlc.AcsAxisIDs[5];
stItpAxes.nQ4AxisId := _refNciChannelRef.NcToPlc.AcsAxisIDs[6];
stItpAxes.nQ5AxisId := _refNciChannelRef.NcToPlc.AcsAxisIDs[7];

ItpAxes := stItpAxes;
END_GET
END_PROPERTY

(*
===============================================================
Implementation of Tc2_NCI.ItpResetEx2
===============================================================
*)
METHOD ItpReset   : HRESULT
VAR_INPUT
  Execute         : BOOL;
END_VAR
VAR_INST
  stMsg           : ST_Message;
  nState,
  nStateError     : DINT;

  hr              : HRESULT;
END_VAR

IF NOT Execute
THEN
  nState                    := 0;
  nStateError               := 0;
END_IF

CASE nState OF
  0:
  hr                        := S_FALSE;

  fbReset(bExecute          := FALSE, 
          tTimeOut          := T#1S, 
          sNciToPlc         := _refNciChannelRef.NcToPlc);
 
  IF Execute 
  THEN
    nState                  := 10;
  END_IF
END_CASE
CASE nState OF
  10:
  fbReset(bExecute          := TRUE, 
          tTimeOut          := T#1S, 
          sNciToPlc         := _refNciChannelRef.NcToPlc);

  IF fbReset.bBusy 
  THEN
    hr                      := S_FALSE;
  ELSIF fbReset.bErr 
  THEN
    stMsg.eType             := E_MessageType.eMessageError;
    stMsg.eDevice           := ChannelDevice;
    stMsg.eSubdevice        := e_Subdevice.fbResetItp;
    stMsg.iErrorNumber      := fbReset.nErrId;
    stMsg.sText             := concat('ItpReset Error: ', UDINT_TO_STRING(fbReset.nErrId));
    f_MessageSet(stMsg);

    hr                      := UDINT_TO_DINT(fbReset.nErrId);
    nStateError             := nState;
    nState                  := 99;
  ELSE
    _sProg                  := '';
    nState                  := 100;
  END_IF
END_CASE
CASE nState OF
  100:
  //Done
  hr                         := S_OK;
END_CASE
//Return Result
ItpReset:= hr;
END_METHOD

(*
===============================================================
Implementation of Tc2_NCI.ItpLoadProgEx
===============================================================
*)
METHOD LoadProg   : HRESULT
VAR_INPUT
  Execute         : BOOL;
END_VAR
VAR_INST
  stMsg           : ST_Message;
  nState,
  nStateError     : DINT;

  hr              : HRESULT;
END_VAR

IF NOT Execute
THEN
  nState                            := 0;
  nStateError                       := 0;
END_IF

CASE nState OF
  0:
    hr                              := S_FALSE;

    fbLoadProg(sNciToPlc            := _refNciChannelRef.NcToPlc, 
               bExecute             := FALSE, 
               sPrg                 := _sProg, 
               nLength              := TO_UDINT(LEN(_sProg)));
    IF Execute
    THEN
      nState := 10;
    END_IF
END_CASE
CASE nState OF
  10:
    fbLoadProg(sNciToPlc            := _refNciChannelRef.NcToPlc, 
               bExecute             := TRUE, 
               sPrg                 := _sProg, 
               nLength              := TO_UDINT(LEN(_sProg)));
  
    IF fbLoadProg.bErr
    THEN
      stMsg.eType                   := E_MessageType.eMessageError;
      stMsg.eDevice                 := ChannelDevice;
      stMsg.eSubdevice              := e_Subdevice.fbLoadProg;
      stMsg.iErrorNumber            := fbLoadProg.nErrId;
      stMsg.sText                   := concat('LoadProg Error: ', TO_STRING(fbLoadProg.nErrId));
      f_MessageSet(stMsg);

      hr                            := TO_DINT(fbLoadProg.nErrId);

      nState                        := 99;
   
    ELSIF NOT fbLoadProg.bBusy
    THEN
      nState                        := 100;

      stMsg.eType                   := E_MessageType.eMessageInfo;
      stMsg.eDevice                 := ChannelDevice;
      stMsg.eSubdevice              := e_Subdevice.fbLoadProg;
      stMsg.iErrorNumber            := fbLoadProg.nErrId;
      stMsg.sText                   := concat('LoadProg Done: ', fbLoadProg.sPrg);
      f_MessageSet(stMsg);
    END_IF
END_CASE
CASE nState OF
  100:
    //Done
    hr                              := S_OK;
END_CASE
//Return Result
LoadProg:= hr;
END_METHOD

(*
===============================================================
M-Function
===============================================================
*)
PROPERTY MFunc : INT
GET

MFunc := TO_INT(_refNciChannelRef.NcToPlc.HskMFuncNo);
END_GET
END_PROPERTY

PROPERTY Override : LREAL
GET
Override := Tc2_NCI.ItpGetOverridePercent(_refNciChannelRef.PlcToNc);
END_GET
SET
Tc2_NCI.ItpSetOverridePercent(Override, _refNciChannelRef.PlcToNc);
END_SET
END_PROPERTY

(*
===============================================================
actual path velo [Units/s]
===============================================================
*)
PROPERTY PathVelo : LREAL
GET

PathVelo := _refNciChannelRef.NcToPlc.PathVelo;
END_GET
END_PROPERTY

PROPERTY pNciChannelRef : POINTER TO ST_NciChannel_Ref
GET
pNciChannelRef := ADR(_refNciChannelRef);
END_GET
END_PROPERTY

(*
===============================================================
G-Code Program Name (sFilePath)
===============================================================
*)
PROPERTY Prog : STRING(255)
GET
Prog:=_sProg;
END_GET
SET
_sProg:=Prog;
END_SET
END_PROPERTY

(*
===============================================================
Implementation of Tc2_System.ADSREADEX

  reads actual interpreter G-Code Line
===============================================================
*)
METHOD ReadLine   : HRESULT
VAR_INPUT
  Execute         : BOOL;
END_VAR
//Read G-Code actual Line
VAR_OUTPUT
  ActProgLine     : STRING(100);
END_VAR
VAR_INST
  ReadString      : STRING(100);
  nBlockNo        : UDINT;

  stMsg           : ST_Message;
  nState,
  nStateError     : DINT;

  hr              : HRESULT;
END_VAR

IF NOT Execute
THEN
  nState                    := 0;
  nStateError               := 0;
END_IF

CASE nState OF
  0:
  hr                        := S_FALSE;

  fbReadLine(PORT           := 500, 
             IDXGRP         := 16#2300 + _refNciChannelRef.NcToPlc.ChnId, // + ChannelID
             IDXOFFS        := 16#2000_0001,
             LEN            := SIZEOF(ReadString),
             DESTADDR       := ADR(ReadString), 
             READ           := FALSE);
  
  IF Execute 
  THEN
    nState                  := 10;
    nBlockNo                := _refNciChannelRef.NcToPlc.BlockNo;
  END_IF
END_CASE
CASE nState OF
  10:
  fbReadLine(PORT           := 500, 
             IDXGRP         := 16#2300 + _refNciChannelRef.NcToPlc.ChnId, // + ChannelID
             IDXOFFS        := 16#2000_0001,
             LEN            := SIZEOF(ReadString),
             DESTADDR       := ADR(ReadString), 
             READ           := TRUE);

  IF fbReadLine.ERR
  THEN
    stMsg.eType             := E_MessageType.eMessageError;
    stMsg.eDevice           := ChannelDevice;
    stMsg.eSubdevice        := e_Subdevice.fbReadLine;
    stMsg.iErrorNumber      := fbReadLine.ERRID;
    stMsg.sText             := concat('fbReadLine ADS error: ', TO_STRING(fbReadLine.ERRID));
    f_MessageSet(stMsg);

    nStateError             := nState;
    nState                  := 99;

  ELSIF NOT fbReadLine.BUSY
  THEN
    nState                  := 100;
    ActProgLine             := ReadString;

    stMsg.eType             := E_MessageType.eMessageInfo;
    stMsg.eDevice           := ChannelDevice;
    stMsg.eSubdevice        := e_Subdevice.fbReadLine;
    stMsg.iErrorNumber      := fbReadLine.ERRID;
    stMsg.sText             := CONCAT(CONCAT(CONCAT('ReadLine Done: ', ReadString), ' Lines:'), TO_STRING(fbReadLine.COUNT_R));
    f_MessageSet(stMsg);
  END_IF
END_CASE
CASE nState OF
  100:
  //Done
  hr                        := S_OK;
END_CASE

//Return Result
ReadLine:= hr;
END_METHOD

(*
===============================================================
Implementation of Tc2_NCI.ItpReadRParamsEx

  read R-Parameter(s) from NCI
===============================================================
*)
METHOD ReadRParams : HRESULT
VAR_INPUT
  Execute  : BOOL;
  Addr     : POINTER TO LREAL;  // start adr of rParam array 
  Index    : DINT;              // start index of R[Index] in NCI
  Count    : DINT;              // count of R[index+i] in NCI
END_VAR
VAR_INST
  stMsg           : ST_Message;
  nState,
  nStateError     : DINT;

  hr              : HRESULT;
END_VAR

IF NOT Execute
THEN
  nState                            := 0;
  nStateError                       := 0;
END_IF

CASE nState OF
  0:
  hr                                := S_FALSE;

  fbItpReadRParams( sNciToPlc       := _refNciChannelRef.NcToPlc, 
                    bExecute        := FALSE, 
                    pAddr           := Addr, 
                    nIndex          := Index, 
                    nCount          := Count);
  
  IF Execute 
  THEN
    nState                          := 10;
  END_IF
END_CASE
CASE nState OF
  10:
  fbItpReadRParams( sNciToPlc       := _refNciChannelRef.NcToPlc, 
                    bExecute        := TRUE, 
                    pAddr           := Addr, 
                    nIndex          := Index, 
                    nCount          := Count);

  IF fbItpReadRParams.bErr
  THEN
    stMsg.eType                     := E_MessageType.eMessageError;
    stMsg.eDevice                   := ChannelDevice;
    stMsg.eSubdevice                := e_Subdevice.fbItpReadRParams;
    stMsg.iErrorNumber              := fbItpReadRParams.nErrId;
    stMsg.sText                     := concat('fbItpReadRParams Error: ', 
                                              TO_STRING(fbItpReadRParams.nERRID));
    f_MessageSet(stMsg);

    hr                              := TO_DINT(fbItpReadRParams.nErrId);
    nStateError                     := nState;
    nState                          := 99;

  ELSIF NOT fbItpReadRParams.bBusy
  THEN
    nState                          := 100;

    stMsg.eType                     := E_MessageType.eMessageInfo;
    stMsg.eDevice                   := ChannelDevice;
    stMsg.eSubdevice                := e_Subdevice.fbItpReadRParams;
    stMsg.iErrorNumber              := fbItpReadRParams.nErrId;
    stMsg.sText                     := concat('fbItpReadRParams Done: ', 
                                              TO_STRING(fbItpReadRParams.nCount));
    f_MessageSet(stMsg);
  END_IF
END_CASE
CASE nState OF
  100:
  //Done
  hr                                := S_OK;
END_CASE

//Return Result
ReadRParams:= hr;
END_METHOD

(*
===============================================================
Implementation of Tc2_NCI.ItpStartStopEx

  Start Interpreter
===============================================================
*)
METHOD StartStop : HRESULT
VAR_INPUT
  Start: BOOL;
  Stop: BOOL;
END_VAR
VAR_INST
  stMsg           : ST_Message;
  nState,
  nStateError     : DINT;

  hr              : HRESULT;
END_VAR

fbStartStop(bStart                  := Start, 
            bStop                   := Stop, 
            sNciToPlc               := _refNciChannelRef.NcToPlc);

  
IF fbStartStop.bBusy 
THEN
  hr                                := S_FALSE;

ELSIF fbStartStop.bErr 
THEN
  IF (stMsg.iErrorNumber <> fbStartStop.nErrId)
  THEN
    stMsg.eType                     := E_MessageType.eMessageError;
    stMsg.eDevice                   := ChannelDevice;
    stMsg.eSubdevice                := e_Subdevice.fbStartStopItp;
    stMsg.iErrorNumber              := fbStartStop.nErrId;
    stMsg.sText                     := concat('Start Interpreter ERROR: ', TO_STRING(fbStartStop.nErrId));
    f_MessageSet(stMsg);
  END_IF

  hr                                := UDINT_TO_DINT(fbStartStop.nErrId);
ELSE
  IF Start
  THEN
    stMsg.eType                     := E_MessageType.eMessageInfo;
    stMsg.eDevice                   := ChannelDevice;
    stMsg.eSubdevice                := e_Subdevice.fbStartStopItp;
    stMsg.iErrorNumber              := 0;
    stMsg.sText                     := concat('Start file: ', _sProg);
    f_MessageSet(stMsg);

  ELSIF Stop
  THEN
    stMsg.eType                     := E_MessageType.eMessageInfo;
    stMsg.eDevice                   := ChannelDevice;
    stMsg.eSubdevice                := e_Subdevice.fbStartStopItp;
    stMsg.iErrorNumber              := 0;
    stMsg.sText                     := concat('Stop file: ', _sProg);
    f_MessageSet(stMsg);
  END_IF
  hr                                := S_OK;
END_IF

//Return Result
StartStop:= hr;
END_METHOD

(*
===============================================================
Implementation of Tc2_NCI.ItpStopOnAfterEStopEx
===============================================================
*)
METHOD StepOnAfterEStop : HRESULT
VAR_INPUT
  Execute: BOOL;
END_VAR
VAR_INST
  stMsg           : ST_Message;
  nState,
  nStateError     : DINT;

  hr              : HRESULT;
END_VAR

IF NOT Execute
THEN
  nState                            := 0;
  nStateError                       := 0;
END_IF

CASE nState OF
  0:
    hr                              := S_FALSE;
    fbStepOnAfterEStop(bExecute     := FALSE, 
                       sNciToPlc    := _refNciChannelRef.NcToPlc);

    IF Execute
    THEN
      nState                        := 10;
    END_IF
END_CASE
CASE nState OF
  10:
    fbStepOnAfterEStop(bExecute     := TRUE, 
                     sNciToPlc      := _refNciChannelRef.NcToPlc);
  
    IF fbStepOnAfterEStop.bErr
    THEN
      stMsg.eType                   := E_MessageType.eMessageError;
      stMsg.eDevice                 := ChannelDevice;
      stMsg.eSubdevice              := e_Subdevice.fbStepOnAfterEStopItp;
      stMsg.iErrorNumber            := fbStepOnAfterEStop.nErrId;
      stMsg.sText                   := concat('StepOn Error: ', TO_STRING(fbStepOnAfterEStop.nErrId));
      f_MessageSet(stMsg);

      hr                            := TO_DINT(fbStepOnAfterEStop.nErrId);

      nState                        := 99;
   
    ELSIF NOT fbStepOnAfterEStop.bBusy
    THEN
      nState                        := 100;

      stMsg.eType                   := E_MessageType.eMessageInfo;
      stMsg.eDevice                 := ChannelDevice;
      stMsg.eSubdevice              := e_Subdevice.fbStepOnAfterEStopItp;
      stMsg.iErrorNumber            := fbStepOnAfterEStop.nErrId;
      stMsg.sText                   := concat('StepOn Group: ', UDINT_TO_STRING(_refNciChannelRef.NcToPlc.GrpId));
      f_MessageSet(stMsg);


      fbStepOnAfterEStop(bExecute   := FALSE, 
                         sNciToPlc  := _refNciChannelRef.NcToPlc);
  
    END_IF
END_CASE
CASE nState OF
  100:
  //Done
  hr                                := S_OK;
END_CASE

//Return Result
StepOnAfterEStop:= hr;
END_METHOD

(*
===============================================================
Implementation of Tc2_NCI.ItpWriteRParamsEx

  write R-Parameter(s) to NCI
===============================================================
*)
METHOD WriteRParams : HRESULT
VAR_INPUT
  Execute : BOOL;
  Addr    : POINTER TO LREAL; // Adresse der Zielvariablen der Daten. 
                              // Dabei werden die Daten direkt ab der angegebenen Adresse von der NC beschrieben  
                              // D.h. nIndex ist nicht als Offset zu pAddr zu sehen. Die Daten befinden sich z.B. 
                              // in einem Array vom Typ LREAL, das vom Anwender definiert werden muss.
  Index   : DINT;
  Count   : DINT;
END_VAR
VAR_INST
  stMsg           : ST_Message;
  nState,
  nStateError     : DINT;

  hr              : HRESULT;
END_VAR

IF NOT Execute
THEN
  nState                            := 0;
  nStateError                       := 0;
END_IF

CASE nState OF
  0:
    hr                              := S_FALSE;

    fbItpWriteRParams(bExecute      := FALSE, 
                      pAddr         := Addr, 
                      nIndex        := Index, 
                      nCount        := Count, 
                      sNciToPlc     := _refNciChannelRef.NcToPlc);
    IF Execute
    THEN
      nState                        := 10;
    END_IF
END_CASE
CASE nState OF
  10:
    fbItpWriteRParams(bExecute      := TRUE, 
                      pAddr         := Addr, 
                      nIndex        := Index, 
                      nCount        := Count, 
                      sNciToPlc     := _refNciChannelRef.NcToPlc);

    IF fbItpWriteRParams.bErr
    THEN
      stMsg.eType                   := E_MessageType.eMessageError;
      stMsg.eDevice                 := ChannelDevice;
      stMsg.eSubdevice              := e_Subdevice.fbItpWriteRParams;
      stMsg.iErrorNumber            := fbItpWriteRParams.nErrId;
      stMsg.sText                   := concat('fbItpWriteRParams Error: ', 
                                                TO_STRING(fbItpWriteRParams.nERRID));
      f_MessageSet(stMsg);
  
      hr                            := TO_DINT(fbItpWriteRParams.nErrId);
      nStateError                   := nState;
      nState                        := 99;
  
    ELSIF NOT fbItpWriteRParams.bBusy
    THEN
      nState                        := 100;
  
      stMsg.eType                   := E_MessageType.eMessageInfo;
      stMsg.eDevice                 := ChannelDevice;
      stMsg.eSubdevice              := e_Subdevice.fbItpWriteRParams;
      stMsg.iErrorNumber            := fbItpWriteRParams.nErrId;
      stMsg.sText                   := concat('fbItpWriteRParams Done: ', 
                                                TO_STRING(fbItpWriteRParams.nCount));
      f_MessageSet(stMsg);
    END_IF
END_CASE
CASE nState OF
  100:
  //Done
  hr                                := S_OK;
END_CASE
//Return Result
WriteRParams:= hr;
END_METHOD

END_FUNCTION_BLOCK

// ---- POUs/_FunctionBlocks/fb_LocalTime.TcPOU
FUNCTION_BLOCK fb_LocalTime
VAR_INPUT

END_VAR
VAR_OUTPUT
  sLocalTime  : STRING;
  dtLocalTime : DT;
END_VAR
VAR
  GetSysTime    : FW_GetSystemTime;
  strFileTime   : T_FILETIME;
END_VAR

GetSysTime(dwTimeLo=> strFileTime.dwLowDateTime, dwTimeHi=> strFileTime.dwHighDateTime);

sLocalTime := SYSTEMTIME_TO_STRING( FILETIME_TO_SYSTEMTIME( strFileTime ) );
dtLocalTime := systemtime_to_dt( FILETIME_TO_SYSTEMTIME( strFileTime ) );

END_FUNCTION_BLOCK

// ---- DOC/DOCUMENTATION.TcPOU
// DOCUMENTATION ONLY
PROGRAM DOCUMENTATION
VAR
END_VAR

;
//---------------------------------------------------------------------------------------------------------------
//
//  HAUD 2023.08.11
//
//
//
//  Documentation TC_Dos_Nci/PLC_OPEN_DRIVE
//
//  - MC and NCI encapsulation for outside use
//  - ADS and cyclic access possible
//  - cyclic interface through TwinCAT mapping (pragmas)
//  - use of compiler defines for software options
//
//-------------------------------------------------------------
//  - cyclic interface to NC
//-------------------------------------------------------------
//    - GVL_AXIS_CTRL.gfbAxisController[].fbAxis.pAxisRef
//    - GVL_NCI.gfbNciCtrl[1]._fbNciChannel._refNciChannelRef
//
//-------------------------------------------------------------
//  - PTP interface to outside world
//-------------------------------------------------------------
//    - GVL_AXIS_CTRL.gstAxisControl - %Q* and %I* cyclic data
//    - GVL_AXIS_CTRL.gstAxisControl : ST_AxisController
//
//  TYPE ST_AxisController :
//  STRUCT
//
//  {IF defined (AXIS_MAP)}
//    {info 'mapped control'}
//    ToPlc    AT %I* : ST_In;
//    FromPlc  AT %Q* : ST_Out;
//  {ELSE}
//    {info 'local control'}
//    ToPlc    : ST_In;
//    FromPlc  : ST_Out;
//  {END_IF}
//
//  END_STRUCT
//  END_TYPE
//
//
//  {attribute 'pack_mode' := '2'}
//  TYPE ST_In :
//  STRUCT
//    bFastStop         : BIT;  // Fast stop function of NC with mapped input
//    byAxisFuncPara    : BYTE; // additional parameter for Axis Function; e.g. used for AxisIndex on GearIn
//    uiAxisFunctionReq : e_AxisFunction; // selected function for axis 
//    rSetPos           : LREAL;
//    rSetVelo          : LREAL;
//    rOverride         : LREAL;
//    rAcc              : LREAL;
//    rDec              : LREAL;
//    iDirection        : INT;
//  END_STRUCT
//  END_TYPE
//
//
//  TYPE e_AxisFunction :
//  (
//    AXIS_DISABLE,
//    AXIS_IDLE := 1,
//    AXIS_ENABLE := 10,
//    AXIS_HOME,
//    AXIS_MOVE_POS,
//    AXIS_MOVE_VELO,
//    AXIS_RESET,
//    AXIS_HALT,
//    AXIS_STOP,
//
//    AXIS_MOVE_BUFFER := 20,
//    AXIS_MOVE_BUFFER_VELO,
//    AXIS_WRITE_BUFFER_MODE,
//
//    AXIS_PARAMETER   := 30, // axis function for reading and writing parameter
//
//
//    AXIS_GEAR_IN    := 50,
//    AXIS_GEAR_OUT,
//    AXIS_GEAR_IN_MULTIMASTER,
//    
//    AXIS_SS1_STOP   :=  99,
//    AXIS_BUSY       := 100,
//    AXIS_STARTUP    := 200,
//    AXIS_DONE       := 1000,
//
//    ERROR           := 9000
//  )UINT;
//  END_TYPE
//
//
//
//-------------------------------------------------------------
//  - NCI interface to outside world
//-------------------------------------------------------------
//
//  - cyclic ctrl interface for starting NCI functions
//      GVL_NCI.gstChannelCtrl  - command struct
//      GVL_NCI.gstChannelState - status struct
//
//  - config structs required for jobs
//      GVL_NCI.gstAxisConfig   - NC Axis Id for building Group
//      GVL_NCI.gstAxisIndex    - Index in GVL_AXIS_CTRL.gfbAxisController[].fbAxis.pAxisRef
//      GVL_NCI.gsProgName      - Commanded name for *.nc file
//      GVL_NCI.gsProgNameActive- active or last *.nc file
//      GVL_NCI.gstRParameter   - array of lreals to use on R Parameter Range (max 10 consecutive entries)
//
//  - available commands:
//
//  {attribute 'qualified_only'}
//  {attribute 'to_string'}
//  TYPE e_Ctrl_NciCommand :
//  (
//    NO_NCI            := -10,
//    NO_AXIS_GROUP     := -2,
//    NO_AXIS_INDEX     := -1,
//    NO_INIT,
//    INIT,
//    IDLE,
//    RESET,
//    LOAD_PROG,
//    FEED_TABLE,
//    BUILD_GROUP,
//    CLEAR_GROUP,
//
//    START         := 10,
//    STOP,
//    STO_STOP,
//    RESTART_STEP_ON,
//
//    M_FUNC_QUIT   := 20,
//
//    READ_R_PARA   := 30,
//    WRITE_R_PARA  := 40,
//
//    CMD_BUSY      := 100,
//    CMD_DONE      := 1000,
//    CMD_ERROR     := 9000
//  )DINT;
//  END_TYPE
//
//
//---------------------------------------------------------------------------------------------------------------
// This SOFTWARE is provided as an Exemple by THE PROVIDER "as is" and "with all faults." THE PROVIDER makes no 
// representations or warranties of any kind concerning the safety, suitability, lack of viruses, inaccuracies, 
// typographical errors, or other harmful components of this SOFTWARE. There are inherent dangers in the use of 
// any software, and you are solely responsible for determining whether this SOFTWARE is compatible with your 
// equipment and other software installed on your equipment. You are also solely responsible for the protection 
// of your equipment and backup of your data, and THE PROVIDER will not be liable for any damages you may suffer 
// in connection with using, modifying, or distributing this SOFTWARE.
//---------------------------------------------------------------------------------------------------------------

END_PROGRAM

// ---- POUs/Functions/f_DelBit64.TcPOU
FUNCTION f_DelBit64 : LWORD
VAR_INPUT
  inVal   : LWORD;
  bitNo   : INT;
END_VAR
VAR
  wConst : LWORD := 1;
END_VAR

IF ( inVal AND SHL( wConst,INT_TO_SINT(bitNo) MOD 64 ) ) > 0 THEN
  f_DelBit64 := inVal XOR (SHL( wConst,INT_TO_SINT(bitNo) MOD 64 ));
ELSE
  f_DelBit64 := inVal;
END_IF

END_FUNCTION

// ---- POUs/Functions/f_GetBit64.TcPOU
FUNCTION f_GetBit64 : bool
VAR_INPUT
	lwIn			: LWORD;
	bitNo			: INT;
END_VAR
VAR
	lwConst		: LWORD := 1;
END_VAR

IF ( lwIn AND SHL( lwConst,INT_TO_SINT(bitNo) MOD 64 ) ) > 0
THEN
	f_GetBit64 := TRUE;
ELSE
	f_GetBit64 := FALSE;
END_IF

END_FUNCTION

// ---- POUs/Functions/f_Setbit64.TcPOU
FUNCTION f_Setbit64 : LWORD
VAR_INPUT
  inVal   : LWORD;
  bitNo   : INT;
END_VAR
VAR
  wConst  : LWORD := 1;
END_VAR

f_Setbit64 := inVal OR SHL( wConst,INT_TO_SINT(bitNo) MOD 64 );

END_FUNCTION

// ---- POUs/_FunctionBlocks/cam/fb_Camming.TcPOU
FUNCTION_BLOCK fb_Camming
VAR_INPUT
END_VAR
VAR_OUTPUT
END_VAR
VAR
  fbCamIn       : Tc2_MC2_Camming.MC_CamIn_V2;
  fbCamOut      : Tc2_MC2_Camming.MC_CamOut;

END_VAR

END_FUNCTION_BLOCK

// ---- POUs/_FunctionBlocks/cam/fb_Camming_Empty.TcPOU
FUNCTION_BLOCK fb_Camming_Empty
VAR_INPUT
END_VAR
VAR_OUTPUT
  Error   : BOOL;
END_VAR
VAR
END_VAR

END_FUNCTION_BLOCK

// ---- POUs/_FunctionBlocks/fb_Blink.TcPOU
FUNCTION_BLOCK fb_Blink
VAR_INPUT
	tLowTime		: TIME;
	tCycleTime	: TIME;
END_VAR
VAR_OUTPUT
	bCycle			: BOOL;
END_VAR
VAR
	tonLowTime		: TON;
	tofCycleTime	: TOF;
END_VAR

tonLowTime(IN:=(NOT tofCycleTime.Q), PT:= tLowTime);
tofCycleTime(IN:=(tonLowTime.Q), PT:= tCycleTime);

bCycle := tofCycleTime.Q;

END_FUNCTION_BLOCK

// ---- GlobalTextList.TcGTLO
TEXTLIST GlobalTextList
  487 = 'eDevice'
  902 = 'Einheit'
  982 = 'eSubdevice'
  872 = 'eType'
  666 = 'Frequency: %s'
  231 = 'iErrorNumber'
  903 = 'Meldung ID'
  94 = 'QUIT'
  901 = 'Station'
  639 = 'sText'
  448 = 'TargetCounter: %s'
  312 = 'tTime'
  900 = 'Type'
  971 = 'Write to file'
  904 = 'Zeitstempel'
END_TEXTLIST

